LIN {X 0,Y 255.719,Z 484.142,A -85,B 0,C 180,E1 -18832.417,E2 -18832.417} C_VEL
LIN {X 0,Y 257.097,Z 472.751,A -85,B 0,C 180,E1 -18833.566,E2 -18833.566} C_VEL
LIN {X 0,Y 258.388,Z 459.153,A -85,B 0,C 180,E1 -18834.561,E2 -18834.561} C_VEL
LIN {X 0,Y 259.209,Z 446.518,A -85,B 0,C 180,E1 -18835.173,E2 -18835.173} C_VEL
LIN {X 0,Y 260.998,Z 385.807,A -85,B 0,C 180,E1 -18836.837,E2 -18836.837} C_VEL
LIN {X 0,Y 256.391,Z 351.056,A -85,B 0,C 180,E1 -18838.294,E2 -18838.294} C_VEL
LIN {X 0,Y 251.982,Z 338.318,A -85,B 0,C 180,E1 -18839.157,E2 -18839.157} C_VEL
LIN {X 0,Y 250.109,Z 329.208,A -85,B 0,C 180,E1 -18842.542,E2 -18842.542} C_VEL
LIN {X 0,Y 249.068,Z 324.462,A -85,B 0,C 180,E1 -18844.447,E2 -18844.447} C_VEL
LIN {X 0,Y 249.006,Z 324.47,A -85,B 0,C 180,E1 -18848.386,E2 -18848.386} C_VEL
LIN {X 0,Y 248.98,Z 324.473,A -85,B 0,C 180,E1 -18852.785,E2 -18852.785} C_VEL
LIN {X 0,Y 249.014,Z 324.467,A -85,B 0,C 180,E1 -18857.362,E2 -18857.362} C_VEL
LIN {X 0,Y 249.031,Z 324.461,A -85,B 0,C 180,E1 -18861.62,E2 -18861.62} C_VEL
LIN {X 0,Y 249.048,Z 324.46,A -85,B 0,C 180,E1 -18865.64,E2 -18865.64} C_VEL
LIN {X 0,Y 249.008,Z 324.466,A -85,B 0,C 180,E1 -18869.467,E2 -18869.467} C_VEL
LIN {X 0,Y 249.046,Z 324.462,A -85,B 0,C 180,E1 -18873.159,E2 -18873.159} C_VEL
LIN {X 0,Y 249.061,Z 324.459,A -85,B 0,C 180,E1 -18876.73,E2 -18876.73} C_VEL
LIN {X 0,Y 249.083,Z 324.443,A -85,B 0,C 180,E1 -18880.209,E2 -18880.209} C_VEL
LIN {X 0,Y 249.182,Z 324.446,A -85,B 0,C 180,E1 -18883.617,E2 -18883.617} C_VEL
LIN {X 0,Y 249.218,Z 324.438,A -85,B 0,C 180,E1 -18886.961,E2 -18886.961} C_VEL
LIN {X 0,Y 249.446,Z 324.399,A -85,B 0,C 180,E1 -18891.901,E2 -18891.901} C_VEL
LIN {X 0,Y 249.28,Z 324.429,A -85,B 0,C 180,E1 -18895.148,E2 -18895.148} C_VEL
LIN {X 0,Y 249.668,Z 324.38,A -85,B 0,C 180,E1 -18898.387,E2 -18898.387} C_VEL
LIN {X 0,Y 249.67,Z 324.37,A -85,B 0,C 180,E1 -18901.613,E2 -18901.613} C_VEL
LIN {X 0,Y 249.429,Z 324.411,A -85,B 0,C 180,E1 -18906.582,E2 -18906.582} C_VEL
LIN {X 0,Y 249.348,Z 324.422,A -85,B 0,C 180,E1 -18909.736,E2 -18909.736} C_VEL
LIN {X 0,Y 249.176,Z 324.427,A -85,B 0,C 180,E1 -18914.705,E2 -18914.705} C_VEL
LIN {X 0,Y 249.107,Z 324.445,A -85,B 0,C 180,E1 -18918.079,E2 -18918.079} C_VEL
LIN {X 0,Y 249.084,Z 324.456,A -85,B 0,C 180,E1 -18921.518,E2 -18921.518} C_VEL
LIN {X 0,Y 249.09,Z 324.445,A -85,B 0,C 180,E1 -18925.46,E2 -18925.46} C_VEL
LIN {X 0,Y 249.04,Z 324.447,A -85,B 0,C 180,E1 -18928.973,E2 -18928.973} C_VEL
LIN {X 0,Y 249.031,Z 324.459,A -85,B 0,C 180,E1 -18932.425,E2 -18932.425} C_VEL
LIN {X 0,Y 249.033,Z 324.454,A -85,B 0,C 180,E1 -18936.344,E2 -18936.344} C_VEL
LIN {X 0,Y 249.009,Z 324.459,A -85,B 0,C 180,E1 -18940.477,E2 -18940.477} C_VEL
LIN {X 0,Y 248.998,Z 324.464,A -85,B 0,C 180,E1 -18944.88,E2 -18944.88} C_VEL
LIN {X 0,Y 249.012,Z 324.455,A -85,B 0,C 180,E1 -18947.36,E2 -18947.36} C_VEL
LIN {X 0,Y 249.026,Z 324.464,A -85,B 0,C 180,E1 -18951.618,E2 -18951.618} C_VEL
LIN {X 0,Y 249.045,Z 324.453,A -85,B 0,C 180,E1 -18955.638,E2 -18955.638} C_VEL
LIN {X 0,Y 249.005,Z 324.465,A -85,B 0,C 180,E1 -18959.465,E2 -18959.465} C_VEL
LIN {X 0,Y 249.045,Z 324.462,A -85,B 0,C 180,E1 -18963.158,E2 -18963.158} C_VEL
LIN {X 0,Y 249.061,Z 324.463,A -85,B 0,C 180,E1 -18966.729,E2 -18966.729} C_VEL
LIN {X 0,Y 249.105,Z 324.457,A -85,B 0,C 180,E1 -18970.21,E2 -18970.21} C_VEL
LIN {X 0,Y 249.258,Z 324.58,A -85,B 0,C 180,E1 -18974.147,E2 -18974.147} C_VEL
LIN {X 0,Y 249.54,Z 325.958,A -85,B 0,C 180,E1 -18974.698,E2 -18974.698} C_VEL
LIN {X 0,Y 257.53,Z 346.854,A -85,B 0,C 180,E1 -18976.149,E2 -18976.149} C_VEL
LIN {X 0,Y 260.689,Z 356.803,A -85,B 0,C 180,E1 -18976.741,E2 -18976.741} C_VEL
LIN {X 0,Y 261.615,Z 362.917,A -85,B 0,C 180,E1 -18977.005,E2 -18977.005} C_VEL
LIN {X 0,Y 259.361,Z 433.833,A -85,B 0,C 180,E1 -18978.943,E2 -18978.943} C_VEL
LIN {X 0,Y 258.474,Z 447.221,A -85,B 0,C 180,E1 -18979.621,E2 -18979.621} C_VEL
LIN {X 0,Y 257.42,Z 459.695,A -85,B 0,C 180,E1 -18980.571,E2 -18980.571} C_VEL
LIN {X 0,Y 256.267,Z 470.812,A -85,B 0,C 180,E1 -18981.72,E2 -18981.72} C_VEL
LIN {X 0,Y 254.576,Z 482.837,A -85,B 0,C 180,E1 -18983.324,E2 -18983.324} C_VEL
LIN {X 0,Y 252.924,Z 493.895,A -85,B 0,C 180,E1 -18985.217,E2 -18985.217} C_VEL
LIN {X 0,Y 251.319,Z 503.079,A -85,B 0,C 180,E1 -18987.194,E2 -18987.194} C_VEL
LIN {X 0,Y 249.795,Z 512.013,A -85,B 0,C 180,E1 -18989.596,E2 -18989.596} C_VEL
LIN {X 0,Y 248.687,Z 519.181,A -85,B 0,C 180,E1 -18992.023,E2 -18992.023} C_VEL
LIN {X 0,Y 247.943,Z 524.03,A -85,B 0,C 180,E1 -18994.062,E2 -18994.062} C_VEL
LIN {X 0,Y 247.436,Z 528.724,A -85,B 0,C 180,E1 -18996.522,E2 -18996.522} C_VEL
LIN {X 0,Y 247.001,Z 532.318,A -85,B 0,C 180,E1 -18999.002,E2 -18999.002} C_VEL
LIN {X 0,Y 246.706,Z 534.889,A -85,B 0,C 180,E1 -19001.501,E2 -19001.501} C_VEL
LIN {X 0,Y 246.684,Z 536.663,A -85,B 0,C 180,E1 -19004.385,E2 -19004.385} C_VEL
LIN {X 0,Y 246.768,Z 537.151,A -85,B 0,C 180,E1 -19006.545,E2 -19006.545} C_VEL
LIN {X 0,Y 246.969,Z 537.091,A -85,B 0,C 180,E1 -19008.24,E2 -19008.24} C_VEL
LIN {X 0,Y 247.414,Z 536.36,A -85,B 0,C 180,E1 -19010.383,E2 -19010.383} C_VEL
LIN {X 0,Y 248.3,Z 534.267,A -85,B 0,C 180,E1 -19013.343,E2 -19013.343} C_VEL
LIN {X 0,Y 249.262,Z 531.781,A -85,B 0,C 180,E1 -19015.546,E2 -19015.546} C_VEL
LIN {X 0,Y 251.01,Z 527.278,A -85,B 0,C 180,E1 -19018.421,E2 -19018.421} C_VEL
LIN {X 0,Y 253.289,Z 520.981,A -85,B 0,C 180,E1 -19021.316,E2 -19021.316} C_VEL
LIN {X 0,Y 255.771,Z 513.958,A -85,B 0,C 180,E1 -19023.778,E2 -19023.778} C_VEL
LIN {X 0,Y 258.049,Z 506.62,A -85,B 0,C 180,E1 -19025.84,E2 -19025.84} C_VEL
LIN {X 0,Y 260.777,Z 497.786,A -85,B 0,C 180,E1 -19027.813,E2 -19027.813} C_VEL
LIN {X 0,Y 263.289,Z 488.607,A -85,B 0,C 180,E1 -19029.459,E2 -19029.459} C_VEL
LIN {X 0,Y 265.977,Z 477.163,A -85,B 0,C 180,E1 -19031.091,E2 -19031.091} C_VEL
LIN {X 0,Y 268.366,Z 465.176,A -85,B 0,C 180,E1 -19032.401,E2 -19032.401} C_VEL
LIN {X 0,Y 270.302,Z 452.398,A -85,B 0,C 180,E1 -19033.432,E2 -19033.432} C_VEL
LIN {X 0,Y 271.66,Z 439.162,A -85,B 0,C 180,E1 -19034.19,E2 -19034.19} C_VEL
LIN {X 0,Y 272.593,Z 424.235,A -85,B 0,C 180,E1 -19034.673,E2 -19034.673} C_VEL
LIN {X 0,Y 274.789,Z 373.279,A -85,B 0,C 180,E1 -19035.986,E2 -19035.986} C_VEL
LIN {X 0,Y 268.616,Z 359.848,A -85,B 0,C 180,E1 -19037.452,E2 -19037.452} C_VEL
LIN {X 0,Y 261.644,Z 346.658,A -85,B 0,C 180,E1 -19039.165,E2 -19039.165} C_VEL
LIN {X 0,Y 254.22,Z 334.263,A -85,B 0,C 180,E1 -19041.093,E2 -19041.093} C_VEL
LIN {X 0,Y 251.4,Z 329.949,A -85,B 0,C 180,E1 -19041.857,E2 -19041.857} C_VEL
LIN {X 0,Y 249.757,Z 326.866,A -85,B 0,C 180,E1 -19042.358,E2 -19042.358} C_VEL
LIN {X 0,Y 249.039,Z 324.465,A -85,B 0,C 180,E1 -19043.745,E2 -19043.745} C_VEL
LIN {X 0,Y 249.025,Z 324.45,A -85,B 0,C 180,E1 -19047.847,E2 -19047.847} C_VEL
LIN {X 0,Y 249.04,Z 324.458,A -85,B 0,C 180,E1 -19051.332,E2 -19051.332} C_VEL
LIN {X 0,Y 249.091,Z 324.451,A -85,B 0,C 180,E1 -19054.962,E2 -19054.962} C_VEL
LIN {X 0,Y 249.044,Z 324.455,A -85,B 0,C 180,E1 -19058.626,E2 -19058.626} C_VEL
LIN {X 0,Y 249.15,Z 324.446,A -85,B 0,C 180,E1 -19063.616,E2 -19063.616} C_VEL
LIN {X 0,Y 249.209,Z 324.441,A -85,B 0,C 180,E1 -19068.615,E2 -19068.615} C_VEL
LIN {X 0,Y 249.405,Z 324.401,A -85,B 0,C 180,E1 -19071.901,E2 -19071.901} C_VEL
LIN {X 0,Y 249.243,Z 324.433,A -85,B 0,C 180,E1 -19075.148,E2 -19075.148} C_VEL
LIN {X 0,Y 249.621,Z 324.384,A -85,B 0,C 180,E1 -19078.973,E2 -19078.973} C_VEL
LIN {X 0,Y 249.649,Z 324.372,A -85,B 0,C 180,E1 -19081.614,E2 -19081.614} C_VEL
LIN {X 0,Y 249.343,Z 324.416,A -85,B 0,C 180,E1 -19085.947,E2 -19085.947} C_VEL
LIN {X 0,Y 248.769,Z 324.485,A -85,B 0,C 180,E1 -19087.294,E2 -19087.294} C_VEL
LIN {X 0,Y 247.167,Z 324.688,A -85,B 0,C 180,E1 -19088.616,E2 -19088.616} C_VEL
LIN {X 0,Y 243.282,Z 325.174,A -85,B 0,C 180,E1 -19091.274,E2 -19091.274} C_VEL
LIN {X 0,Y 242.198,Z 325.297,A -85,B 0,C 180,E1 -19092.665,E2 -19092.665} C_VEL
LIN {X 0,Y 242.121,Z 325.305,A -85,B 0,C 180,E1 -19093.137,E2 -19093.137} C_VEL
LIN {X 0,Y 242.106,Z 325.316,A -85,B 0,C 180,E1 -19096.876,E2 -19096.876} C_VEL
LIN {X 0,Y 242.012,Z 325.332,A -85,B 0,C 180,E1 -19101.683,E2 -19101.683} C_VEL
LIN {X 0,Y 241.987,Z 325.34,A -85,B 0,C 180,E1 -19105.827,E2 -19105.827} C_VEL
LIN {X 0,Y 241.963,Z 325.347,A -85,B 0,C 180,E1 -19109.59,E2 -19109.59} C_VEL
LIN {X 0,Y 241.973,Z 325.345,A -85,B 0,C 180,E1 -19113.494,E2 -19113.494} C_VEL
LIN {X 0,Y 241.959,Z 325.345,A -85,B 0,C 180,E1 -19117.588,E2 -19117.588} C_VEL
LIN {X 0,Y 241.901,Z 325.336,A -85,B 0,C 180,E1 -19121.931,E2 -19121.931} C_VEL
LIN {X 0,Y 241.928,Z 325.445,A -85,B 0,C 180,E1 -19124.566,E2 -19124.566} C_VEL
LIN {X 0,Y 244.093,Z 332.594,A -85,B 0,C 180,E1 -19128.533,E2 -19128.533} C_VEL
LIN {X 0,Y 245.363,Z 336.886,A -85,B 0,C 180,E1 -19130.739,E2 -19130.739} C_VEL
LIN {X 0,Y 247.923,Z 341.395,A -85,B 0,C 180,E1 -19131.498,E2 -19131.498} C_VEL
LIN {X 0,Y 252.243,Z 349.01,A -85,B 0,C 180,E1 -19132.724,E2 -19132.724} C_VEL
LIN {X 0,Y 258.272,Z 360.24,A -85,B 0,C 180,E1 -19134.35,E2 -19134.35} C_VEL
LIN {X 0,Y 265.204,Z 375.094,A -85,B 0,C 180,E1 -19136.145,E2 -19136.145} C_VEL
LIN {X 0,Y 266.211,Z 378.364,A -85,B 0,C 180,E1 -19136.431,E2 -19136.431} C_VEL
LIN {X 0,Y 268.448,Z 392.441,A -85,B 0,C 180,E1 -19137.285,E2 -19137.285} C_VEL
LIN {X 0,Y 265.992,Z 446.475,A -85,B 0,C 180,E1 -19138.744,E2 -19138.744} C_VEL
LIN {X 0,Y 264.593,Z 460.076,A -85,B 0,C 180,E1 -19139.385,E2 -19139.385} C_VEL
LIN {X 0,Y 262.629,Z 472.258,A -85,B 0,C 180,E1 -19140.218,E2 -19140.218} C_VEL
LIN {X 0,Y 260.301,Z 484.181,A -85,B 0,C 180,E1 -19141.366,E2 -19141.366} C_VEL
LIN {X 0,Y 257.528,Z 495.6,A -85,B 0,C 180,E1 -19142.801,E2 -19142.801} C_VEL
LIN {X 0,Y 254.771,Z 505.898,A -85,B 0,C 180,E1 -19144.469,E2 -19144.469} C_VEL
LIN {X 0,Y 252.107,Z 514.351,A -85,B 0,C 180,E1 -19146.16,E2 -19146.16} C_VEL
LIN {X 0,Y 249.473,Z 522.167,A -85,B 0,C 180,E1 -19148.084,E2 -19148.084} C_VEL
LIN {X 0,Y 246.92,Z 529.825,A -85,B 0,C 180,E1 -19150.463,E2 -19150.463} C_VEL
LIN {X 0,Y 244.37,Z 536.91,A -85,B 0,C 180,E1 -19153.288,E2 -19153.288} C_VEL
LIN {X 0,Y 242.596,Z 541.655,A -85,B 0,C 180,E1 -19155.746,E2 -19155.746} C_VEL
LIN {X 0,Y 241.34,Z 545.309,A -85,B 0,C 180,E1 -19158.24,E2 -19158.24} C_VEL
LIN {X 0,Y 240.725,Z 547.212,A -85,B 0,C 180,E1 -19159.913,E2 -19159.913} C_VEL
LIN {X 0,Y 240.275,Z 548.673,A -85,B 0,C 180,E1 -19161.592,E2 -19161.592} C_VEL
LIN {X 0,Y 239.802,Z 550.385,A -85,B 0,C 180,E1 -19164.957,E2 -19164.957} C_VEL
LIN {X 0,Y 239.763,Z 550.671,A -85,B 0,C 180,E1 -19166.641,E2 -19166.641} C_VEL
LIN {X 0,Y 239.832,Z 550.555,A -85,B 0,C 180,E1 -19168.322,E2 -19168.322} C_VEL
LIN {X 0,Y 239.915,Z 550.015,A -85,B 0,C 180,E1 -19170.002,E2 -19170.002} C_VEL
LIN {X 0,Y 239.868,Z 549.078,A -85,B 0,C 180,E1 -19171.68,E2 -19171.68} C_VEL
LIN {X 0,Y 239.807,Z 547.737,A -85,B 0,C 180,E1 -19173.362,E2 -19173.362} C_VEL
LIN {X 0,Y 239.907,Z 544.883,A -85,B 0,C 180,E1 -19175.886,E2 -19175.886} C_VEL
LIN {X 0,Y 240.201,Z 540.977,A -85,B 0,C 180,E1 -19178.414,E2 -19178.414} C_VEL
LIN {X 0,Y 240.76,Z 535.915,A -85,B 0,C 180,E1 -19180.939,E2 -19180.939} C_VEL
LIN {X 0,Y 241.624,Z 529.527,A -85,B 0,C 180,E1 -19183.457,E2 -19183.457} C_VEL
LIN {X 0,Y 242.956,Z 521.508,A -85,B 0,C 180,E1 -19185.952,E2 -19185.952} C_VEL
LIN {X 0,Y 244.419,Z 513.328,A -85,B 0,C 180,E1 -19188.007,E2 -19188.007} C_VEL
LIN {X 0,Y 245.93,Z 503.3,A -85,B 0,C 180,E1 -19190.057,E2 -19190.057} C_VEL
LIN {X 0,Y 247.736,Z 492.021,A -85,B 0,C 180,E1 -19191.862,E2 -19191.862} C_VEL
LIN {X 0,Y 249.346,Z 480.953,A -85,B 0,C 180,E1 -19193.242,E2 -19193.242} C_VEL
LIN {X 0,Y 250.815,Z 468.678,A -85,B 0,C 180,E1 -19194.414,E2 -19194.414} C_VEL
LIN {X 0,Y 251.969,Z 455.818,A -85,B 0,C 180,E1 -19195.285,E2 -19195.285} C_VEL
LIN {X 0,Y 252.75,Z 442.198,A -85,B 0,C 180,E1 -19195.864,E2 -19195.864} C_VEL
LIN {X 0,Y 254.347,Z 386.316,A -85,B 0,C 180,E1 -19197.418,E2 -19197.418} C_VEL
LIN {X 0,Y 250.029,Z 353.01,A -85,B 0,C 180,E1 -19198.857,E2 -19198.857} C_VEL
LIN {X 0,Y 244.73,Z 338.103,A -85,B 0,C 180,E1 -19199.918,E2 -19199.918} C_VEL
LIN {X 0,Y 242.559,Z 327.821,A -85,B 0,C 180,E1 -19203.902,E2 -19203.902} C_VEL
LIN {X 0,Y 242.024,Z 325.336,A -85,B 0,C 180,E1 -19204.997,E2 -19204.997} C_VEL
LIN {X 0,Y 241.934,Z 325.35,A -85,B 0,C 180,E1 -19209.725,E2 -19209.725} C_VEL
LIN {X 0,Y 241.915,Z 325.355,A -85,B 0,C 180,E1 -19214.207,E2 -19214.207} C_VEL
LIN {X 0,Y 241.939,Z 325.351,A -85,B 0,C 180,E1 -19218.077,E2 -19218.077} C_VEL
LIN {X 0,Y 241.992,Z 325.341,A -85,B 0,C 180,E1 -19222.418,E2 -19222.418} C_VEL
LIN {X 0,Y 241.985,Z 325.342,A -85,B 0,C 180,E1 -19226.508,E2 -19226.508} C_VEL
LIN {X 0,Y 241.984,Z 325.342,A -85,B 0,C 180,E1 -19230.612,E2 -19230.612} C_VEL
LIN {X 0,Y 242.038,Z 325.333,A -85,B 0,C 180,E1 -19234.179,E2 -19234.179} C_VEL
LIN {X 0,Y 242.028,Z 325.329,A -85,B 0,C 180,E1 -19238.316,E2 -19238.316} C_VEL
LIN {X 0,Y 242.121,Z 325.322,A -85,B 0,C 180,E1 -19243.316,E2 -19243.316} C_VEL
LIN {X 0,Y 242.183,Z 325.308,A -85,B 0,C 180,E1 -19248.279,E2 -19248.279} C_VEL
LIN {X 0,Y 242.395,Z 325.274,A -85,B 0,C 180,E1 -19251.664,E2 -19251.664} C_VEL
LIN {X 0,Y 242.241,Z 325.306,A -85,B 0,C 180,E1 -19255.006,E2 -19255.006} C_VEL
LIN {X 0,Y 242.628,Z 325.257,A -85,B 0,C 180,E1 -19258.34,E2 -19258.34} C_VEL
LIN {X 0,Y 242.63,Z 325.245,A -85,B 0,C 180,E1 -19261.659,E2 -19261.659} C_VEL
LIN {X 0,Y 242.407,Z 325.288,A -85,B 0,C 180,E1 -19266.659,E2 -19266.659} C_VEL
LIN {X 0,Y 242.272,Z 325.305,A -85,B 0,C 180,E1 -19270.023,E2 -19270.023} C_VEL
LIN {X 0,Y 242.131,Z 325.302,A -85,B 0,C 180,E1 -19275.143,E2 -19275.143} C_VEL
LIN {X 0,Y 242.046,Z 325.327,A -85,B 0,C 180,E1 -19278.626,E2 -19278.626} C_VEL
LIN {X 0,Y 242.007,Z 325.337,A -85,B 0,C 180,E1 -19282.18,E2 -19282.18} C_VEL
LIN {X 0,Y 242.036,Z 325.321,A -85,B 0,C 180,E1 -19285.82,E2 -19285.82} C_VEL
LIN {X 0,Y 241.972,Z 325.332,A -85,B 0,C 180,E1 -19289.588,E2 -19289.588} C_VEL
LIN {X 0,Y 241.983,Z 325.341,A -85,B 0,C 180,E1 -19293.492,E2 -19293.492} C_VEL
LIN {X 0,Y 241.989,Z 325.325,A -85,B 0,C 180,E1 -19297.581,E2 -19297.581} C_VEL
LIN {X 0,Y 241.94,Z 325.346,A -85,B 0,C 180,E1 -19301.921,E2 -19301.921} C_VEL
LIN {X 0,Y 241.93,Z 325.337,A -85,B 0,C 180,E1 -19306.572,E2 -19306.572} C_VEL
LIN {X 0,Y 241.958,Z 325.346,A -85,B 0,C 180,E1 -19310.28,E2 -19310.28} C_VEL
LIN {X 0,Y 241.987,Z 325.333,A -85,B 0,C 180,E1 -19314.488,E2 -19314.488} C_VEL
LIN {X 0,Y 241.956,Z 325.347,A -85,B 0,C 180,E1 -19318.476,E2 -19318.476} C_VEL
LIN {X 0,Y 241.976,Z 325.344,A -85,B 0,C 180,E1 -19322.307,E2 -19322.307} C_VEL
LIN {X 0,Y 242.039,Z 325.335,A -85,B 0,C 180,E1 -19326.013,E2 -19326.013} C_VEL
LIN {X 0,Y 242.034,Z 325.337,A -85,B 0,C 180,E1 -19329.606,E2 -19329.606} C_VEL
LIN {X 0,Y 242.174,Z 325.41,A -85,B 0,C 180,E1 -19333.616,E2 -19333.616} C_VEL
LIN {X 0,Y 242.324,Z 326.153,A -85,B 0,C 180,E1 -19333.924,E2 -19333.924} C_VEL
LIN {X 0,Y 250.238,Z 346.246,A -85,B 0,C 180,E1 -19335.415,E2 -19335.415} C_VEL
LIN {X 0,Y 254.218,Z 358.37,A -85,B 0,C 180,E1 -19336.181,E2 -19336.181} C_VEL
LIN {X 0,Y 255.039,Z 363.888,A -85,B 0,C 180,E1 -19336.428,E2 -19336.428} C_VEL
LIN {X 0,Y 252.719,Z 434.063,A -85,B 0,C 180,E1 -19338.391,E2 -19338.391} C_VEL
LIN {X 0,Y 251.799,Z 447.489,A -85,B 0,C 180,E1 -19339.088,E2 -19339.088} C_VEL
LIN {X 0,Y 250.757,Z 459.388,A -85,B 0,C 180,E1 -19340.012,E2 -19340.012} C_VEL
LIN {X 0,Y 249.462,Z 471.44,A -85,B 0,C 180,E1 -19341.289,E2 -19341.289} C_VEL
LIN {X 0,Y 247.78,Z 482.955,A -85,B 0,C 180,E1 -19342.867,E2 -19342.867} C_VEL
LIN {X 0,Y 246.116,Z 493.358,A -85,B 0,C 180,E1 -19344.674,E2 -19344.674} C_VEL
LIN {X 0,Y 244.491,Z 502.683,A -85,B 0,C 180,E1 -19346.703,E2 -19346.703} C_VEL
LIN {X 0,Y 242.914,Z 511.712,A -85,B 0,C 180,E1 -19349.17,E2 -19349.17} C_VEL
LIN {X 0,Y 241.731,Z 518.983,A -85,B 0,C 180,E1 -19351.665,E2 -19351.665} C_VEL
LIN {X 0,Y 240.831,Z 524.793,A -85,B 0,C 180,E1 -19354.182,E2 -19354.182} C_VEL
LIN {X 0,Y 240.291,Z 529.359,A -85,B 0,C 180,E1 -19356.717,E2 -19356.717} C_VEL
LIN {X 0,Y 240.001,Z 531.774,A -85,B 0,C 180,E1 -19358.418,E2 -19358.418} C_VEL
LIN {X 0,Y 239.739,Z 533.761,A -85,B 0,C 180,E1 -19360.129,E2 -19360.129} C_VEL
LIN {X 0,Y 239.582,Z 535.318,A -85,B 0,C 180,E1 -19361.848,E2 -19361.848} C_VEL
LIN {X 0,Y 239.605,Z 536.865,A -85,B 0,C 180,E1 -19364.548,E2 -19364.548} C_VEL
LIN {X 0,Y 239.712,Z 537.382,A -85,B 0,C 180,E1 -19367.047,E2 -19367.047} C_VEL
LIN {X 0,Y 239.962,Z 537.232,A -85,B 0,C 180,E1 -19368.792,E2 -19368.792} C_VEL
LIN {X 0,Y 240.379,Z 536.58,A -85,B 0,C 180,E1 -19370.678,E2 -19370.678} C_VEL
LIN {X 0,Y 241.46,Z 534.213,A -85,B 0,C 180,E1 -19374.045,E2 -19374.045} C_VEL
LIN {X 0,Y 242.702,Z 531.284,A -85,B 0,C 180,E1 -19376.574,E2 -19376.574} C_VEL
LIN {X 0,Y 244.455,Z 526.964,A -85,B 0,C 180,E1 -19379.256,E2 -19379.256} C_VEL
LIN {X 0,Y 246.563,Z 521.484,A -85,B 0,C 180,E1 -19381.823,E2 -19381.823} C_VEL
LIN {X 0,Y 249.129,Z 514.543,A -85,B 0,C 180,E1 -19384.345,E2 -19384.345} C_VEL
LIN {X 0,Y 251.503,Z 507.387,A -85,B 0,C 180,E1 -19386.426,E2 -19386.426} C_VEL
LIN {X 0,Y 254.348,Z 498.71,A -85,B 0,C 180,E1 -19388.439,E2 -19388.439} C_VEL
LIN {X 0,Y 257.098,Z 489.107,A -85,B 0,C 180,E1 -19390.219,E2 -19390.219} C_VEL
LIN {X 0,Y 259.74,Z 478.482,A -85,B 0,C 180,E1 -19391.78,E2 -19391.78} C_VEL
LIN {X 0,Y 262.196,Z 466.802,A -85,B 0,C 180,E1 -19393.116,E2 -19393.116} C_VEL
LIN {X 0,Y 264.127,Z 455.272,A -85,B 0,C 180,E1 -19394.117,E2 -19394.117} C_VEL
LIN {X 0,Y 265.681,Z 441.84,A -85,B 0,C 180,E1 -19394.948,E2 -19394.948} C_VEL
LIN {X 0,Y 266.64,Z 428.837,A -85,B 0,C 180,E1 -19395.449,E2 -19395.449} C_VEL
LIN {X 0,Y 269.139,Z 376.062,A -85,B 0,C 180,E1 -19396.815,E2 -19396.815} C_VEL
LIN {X 0,Y 267.651,Z 372.135,A -85,B 0,C 180,E1 -19397.199,E2 -19397.199} C_VEL
LIN {X 0,Y 260.471,Z 357.236,A -85,B 0,C 180,E1 -19399.005,E2 -19399.005} C_VEL
LIN {X 0,Y 253.369,Z 344.62,A -85,B 0,C 180,E1 -19400.873,E2 -19400.873} C_VEL
LIN {X 0,Y 247.499,Z 335.143,A -85,B 0,C 180,E1 -19402.509,E2 -19402.509} C_VEL
LIN {X 0,Y 245.051,Z 331.288,A -85,B 0,C 180,E1 -19403.225,E2 -19403.225} C_VEL
LIN {X 0,Y 242.452,Z 327.124,A -85,B 0,C 180,E1 -19404.058,E2 -19404.058} C_VEL
LIN {X 0,Y 241.996,Z 325.318,A -85,B 0,C 180,E1 -19405.127,E2 -19405.127} C_VEL
LIN {X 0,Y 241.946,Z 325.342,A -85,B 0,C 180,E1 -19408.476,E2 -19408.476} C_VEL
LIN {X 0,Y 241.959,Z 325.347,A -85,B 0,C 180,E1 -19412.307,E2 -19412.307} C_VEL
LIN {X 0,Y 242.013,Z 325.34,A -85,B 0,C 180,E1 -19416.012,E2 -19416.012} C_VEL
LIN {X 0,Y 241.976,Z 325.343,A -85,B 0,C 180,E1 -19419.603,E2 -19419.603} C_VEL
LIN {X 0,Y 242.097,Z 325.322,A -85,B 0,C 180,E1 -19423.324,E2 -19423.324} C_VEL
LIN {X 0,Y 242.143,Z 325.317,A -85,B 0,C 180,E1 -19428.278,E2 -19428.278} C_VEL
LIN {X 0,Y 242.359,Z 325.278,A -85,B 0,C 180,E1 -19431.664,E2 -19431.664} C_VEL
LIN {X 0,Y 242.386,Z 325.289,A -85,B 0,C 180,E1 -19433.34,E2 -19433.34} C_VEL
LIN {X 0,Y 242.597,Z 325.258,A -85,B 0,C 180,E1 -19438.34,E2 -19438.34} C_VEL
LIN {X 0,Y 242.609,Z 325.248,A -85,B 0,C 180,E1 -19441.66,E2 -19441.66} C_VEL
LIN {X 0,Y 242.39,Z 325.278,A -85,B 0,C 180,E1 -19446.66,E2 -19446.66} C_VEL
LIN {X 0,Y 242.259,Z 325.304,A -85,B 0,C 180,E1 -19450.024,E2 -19450.024} C_VEL
LIN {X 0,Y 242.121,Z 325.305,A -85,B 0,C 180,E1 -19453.137,E2 -19453.137} C_VEL
LIN {X 0,Y 241.464,Z 325.396,A -85,B 0,C 180,E1 -19454.525,E2 -19454.525} C_VEL
LIN {X 0,Y 238.549,Z 325.76,A -85,B 0,C 180,E1 -19456.786,E2 -19456.786} C_VEL
LIN {X 0,Y 236.071,Z 326.063,A -85,B 0,C 180,E1 -19458.629,E2 -19458.629} C_VEL
LIN {X 0,Y 235.031,Z 326.203,A -85,B 0,C 180,E1 -19460.061,E2 -19460.061} C_VEL
LIN {X 0,Y 234.96,Z 326.208,A -85,B 0,C 180,E1 -19460.547,E2 -19460.547} C_VEL
LIN {X 0,Y 234.918,Z 326.218,A -85,B 0,C 180,E1 -19464.762,E2 -19464.762} C_VEL
LIN {X 0,Y 234.894,Z 326.217,A -85,B 0,C 180,E1 -19468.602,E2 -19468.602} C_VEL
LIN {X 0,Y 234.935,Z 326.218,A -85,B 0,C 180,E1 -19473.115,E2 -19473.115} C_VEL
LIN {X 0,Y 234.901,Z 326.223,A -85,B 0,C 180,E1 -19476.755,E2 -19476.755} C_VEL
LIN {X 0,Y 234.907,Z 326.217,A -85,B 0,C 180,E1 -19478.937,E2 -19478.937} C_VEL
LIN {X 0,Y 234.846,Z 326.254,A -85,B 0,C 180,E1 -19482.973,E2 -19482.973} C_VEL
LIN {X 0,Y 236.943,Z 333.006,A -85,B 0,C 180,E1 -19486.986,E2 -19486.986} C_VEL
LIN {X 0,Y 238.036,Z 336.737,A -85,B 0,C 180,E1 -19488.961,E2 -19488.961} C_VEL
LIN {X 0,Y 240.812,Z 341.34,A -85,B 0,C 180,E1 -19489.849,E2 -19489.849} C_VEL
LIN {X 0,Y 245.278,Z 348.905,A -85,B 0,C 180,E1 -19491.209,E2 -19491.209} C_VEL
LIN {X 0,Y 250.995,Z 359.266,A -85,B 0,C 180,E1 -19492.859,E2 -19492.859} C_VEL
LIN {X 0,Y 258.542,Z 374.896,A -85,B 0,C 180,E1 -19494.933,E2 -19494.933} C_VEL
LIN {X 0,Y 260.834,Z 380.697,A -85,B 0,C 180,E1 -19495.565,E2 -19495.565} C_VEL
LIN {X 0,Y 262.83,Z 393.388,A -85,B 0,C 180,E1 -19496.365,E2 -19496.365} C_VEL
LIN {X 0,Y 260.35,Z 445.928,A -85,B 0,C 180,E1 -19497.804,E2 -19497.804} C_VEL
LIN {X 0,Y 258.909,Z 459.585,A -85,B 0,C 180,E1 -19498.45,E2 -19498.45} C_VEL
LIN {X 0,Y 256.941,Z 471.451,A -85,B 0,C 180,E1 -19499.261,E2 -19499.261} C_VEL
LIN {X 0,Y 254.514,Z 483.556,A -85,B 0,C 180,E1 -19500.425,E2 -19500.425} C_VEL
LIN {X 0,Y 251.651,Z 495.05,A -85,B 0,C 180,E1 -19501.885,E2 -19501.885} C_VEL
LIN {X 0,Y 248.708,Z 505.414,A -85,B 0,C 180,E1 -19503.574,E2 -19503.574} C_VEL
LIN {X 0,Y 245.652,Z 514.783,A -85,B 0,C 180,E1 -19505.493,E2 -19505.493} C_VEL
LIN {X 0,Y 242.414,Z 523.833,A -85,B 0,C 180,E1 -19507.86,E2 -19507.86} C_VEL
LIN {X 0,Y 239.85,Z 531.143,A -85,B 0,C 180,E1 -19510.309,E2 -19510.309} C_VEL
LIN {X 0,Y 237.582,Z 537.035,A -85,B 0,C 180,E1 -19512.795,E2 -19512.795} C_VEL
LIN {X 0,Y 235.711,Z 541.708,A -85,B 0,C 180,E1 -19515.321,E2 -19515.321} C_VEL
LIN {X 0,Y 234.375,Z 545.296,A -85,B 0,C 180,E1 -19517.885,E2 -19517.885} C_VEL
LIN {X 0,Y 233.724,Z 547.16,A -85,B 0,C 180,E1 -19519.608,E2 -19519.608} C_VEL
LIN {X 0,Y 232.905,Z 549.59,A -85,B 0,C 180,E1 -19523.069,E2 -19523.069} C_VEL
LIN {X 0,Y 232.672,Z 550.483,A -85,B 0,C 180,E1 -19526.538,E2 -19526.538} C_VEL
LIN {X 0,Y 232.743,Z 550.315,A -85,B 0,C 180,E1 -19528.271,E2 -19528.271} C_VEL
LIN {X 0,Y 232.846,Z 549.747,A -85,B 0,C 180,E1 -19530.002,E2 -19530.002} C_VEL
LIN {X 0,Y 232.778,Z 548.78,A -85,B 0,C 180,E1 -19531.732,E2 -19531.732} C_VEL
LIN {X 0,Y 232.759,Z 545.989,A -85,B 0,C 180,E1 -19534.85,E2 -19534.85} C_VEL
LIN {X 0,Y 233.004,Z 541.967,A -85,B 0,C 180,E1 -19537.802,E2 -19537.802} C_VEL
LIN {X 0,Y 233.496,Z 537.227,A -85,B 0,C 180,E1 -19540.406,E2 -19540.406} C_VEL
LIN {X 0,Y 234.502,Z 530.075,A -85,B 0,C 180,E1 -19543.432,E2 -19543.432} C_VEL
LIN {X 0,Y 235.853,Z 522.29,A -85,B 0,C 180,E1 -19546.001,E2 -19546.001} C_VEL
LIN {X 0,Y 237.49,Z 513.193,A -85,B 0,C 180,E1 -19548.378,E2 -19548.378} C_VEL
LIN {X 0,Y 239.01,Z 503.533,A -85,B 0,C 180,E1 -19550.416,E2 -19550.416} C_VEL
LIN {X 0,Y 240.616,Z 493.635,A -85,B 0,C 180,E1 -19552.091,E2 -19552.091} C_VEL
LIN {X 0,Y 242.351,Z 483.078,A -85,B 0,C 180,E1 -19553.501,E2 -19553.501} C_VEL
LIN {X 0,Y 243.946,Z 470.304,A -85,B 0,C 180,E1 -19554.807,E2 -19554.807} C_VEL
LIN {X 0,Y 245.149,Z 457.51,A -85,B 0,C 180,E1 -19555.755,E2 -19555.755} C_VEL
LIN {X 0,Y 246.021,Z 445.318,A -85,B 0,C 180,E1 -19556.34,E2 -19556.34} C_VEL
LIN {X 0,Y 247.789,Z 387.009,A -85,B 0,C 180,E1 -19558.018,E2 -19558.018} C_VEL
LIN {X 0,Y 243.752,Z 355.347,A -85,B 0,C 180,E1 -19559.425,E2 -19559.425} C_VEL
LIN {X 0,Y 238.106,Z 339.877,A -85,B 0,C 180,E1 -19560.541,E2 -19560.541} C_VEL
LIN {X 0,Y 237.468,Z 337.867,A -85,B 0,C 180,E1 -19560.734,E2 -19560.734} C_VEL
LIN {X 0,Y 235.437,Z 328.392,A -85,B 0,C 180,E1 -19564.554,E2 -19564.554} C_VEL
LIN {X 0,Y 234.955,Z 326.215,A -85,B 0,C 180,E1 -19565.521,E2 -19565.521} C_VEL
LIN {X 0,Y 234.916,Z 326.223,A -85,B 0,C 180,E1 -19568.936,E2 -19568.936} C_VEL
LIN {X 0,Y 234.879,Z 326.231,A -85,B 0,C 180,E1 -19574.1,E2 -19574.1} C_VEL
LIN {X 0,Y 234.887,Z 326.228,A -85,B 0,C 180,E1 -19578.832,E2 -19578.832} C_VEL
LIN {X 0,Y 234.923,Z 326.22,A -85,B 0,C 180,E1 -19581.079,E2 -19581.079} C_VEL
LIN {X 0,Y 234.932,Z 326.219,A -85,B 0,C 180,E1 -19585.362,E2 -19585.362} C_VEL
LIN {X 0,Y 234.905,Z 326.223,A -85,B 0,C 180,E1 -19589.428,E2 -19589.428} C_VEL
LIN {X 0,Y 234.975,Z 326.213,A -85,B 0,C 180,E1 -19593.807,E2 -19593.807} C_VEL
LIN {X 0,Y 234.993,Z 326.202,A -85,B 0,C 180,E1 -19598.968,E2 -19598.968} C_VEL
LIN {X 0,Y 235.061,Z 326.2,A -85,B 0,C 180,E1 -19603.092,E2 -19603.092} C_VEL
LIN {X 0,Y 235.115,Z 326.19,A -85,B 0,C 180,E1 -19607.922,E2 -19607.922} C_VEL
LIN {X 0,Y 235.328,Z 326.151,A -85,B 0,C 180,E1 -19611.412,E2 -19611.412} C_VEL
LIN {X 0,Y 235.366,Z 326.156,A -85,B 0,C 180,E1 -19613.14,E2 -19613.14} C_VEL
LIN {X 0,Y 235.587,Z 326.134,A -85,B 0,C 180,E1 -19618.29,E2 -19618.29} C_VEL
LIN {X 0,Y 235.588,Z 326.12,A -85,B 0,C 180,E1 -19621.709,E2 -19621.709} C_VEL
LIN {X 0,Y 235.359,Z 326.165,A -85,B 0,C 180,E1 -19626.86,E2 -19626.86} C_VEL
LIN {X 0,Y 235.219,Z 326.185,A -85,B 0,C 180,E1 -19630.327,E2 -19630.327} C_VEL
LIN {X 0,Y 235.078,Z 326.18,A -85,B 0,C 180,E1 -19635.608,E2 -19635.608} C_VEL
LIN {X 0,Y 234.988,Z 326.211,A -85,B 0,C 180,E1 -19639.207,E2 -19639.207} C_VEL
LIN {X 0,Y 234.95,Z 326.218,A -85,B 0,C 180,E1 -19642.884,E2 -19642.884} C_VEL
LIN {X 0,Y 234.949,Z 326.2,A -85,B 0,C 180,E1 -19646.659,E2 -19646.659} C_VEL
LIN {X 0,Y 234.903,Z 326.214,A -85,B 0,C 180,E1 -19650.571,E2 -19650.571} C_VEL
LIN {X 0,Y 234.93,Z 326.215,A -85,B 0,C 180,E1 -19654.638,E2 -19654.638} C_VEL
LIN {X 0,Y 234.945,Z 326.199,A -85,B 0,C 180,E1 -19658.943,E2 -19658.943} C_VEL
LIN {X 0,Y 234.888,Z 326.225,A -85,B 0,C 180,E1 -19663.485,E2 -19663.485} C_VEL
LIN {X 0,Y 234.883,Z 326.214,A -85,B 0,C 180,E1 -19666.511,E2 -19666.511} C_VEL
LIN {X 0,Y 234.92,Z 326.22,A -85,B 0,C 180,E1 -19671.077,E2 -19671.077} C_VEL
LIN {X 0,Y 234.931,Z 326.21,A -85,B 0,C 180,E1 -19675.36,E2 -19675.36} C_VEL
LIN {X 0,Y 234.902,Z 326.222,A -85,B 0,C 180,E1 -19679.426,E2 -19679.426} C_VEL
LIN {X 0,Y 234.971,Z 326.215,A -85,B 0,C 180,E1 -19683.805,E2 -19683.805} C_VEL
LIN {X 0,Y 234.998,Z 326.215,A -85,B 0,C 180,E1 -19688.967,E2 -19688.967} C_VEL
LIN {X 0,Y 235.121,Z 326.379,A -85,B 0,C 180,E1 -19693.107,E2 -19693.107} C_VEL
LIN {X 0,Y 236.293,Z 329.307,A -85,B 0,C 180,E1 -19693.36,E2 -19693.36} C_VEL
LIN {X 0,Y 242.991,Z 345.81,A -85,B 0,C 180,E1 -19694.65,E2 -19694.65} C_VEL
LIN {X 0,Y 247.745,Z 359.842,A -85,B 0,C 180,E1 -19695.589,E2 -19695.589} C_VEL
LIN {X 0,Y 248.492,Z 365.668,A -85,B 0,C 180,E1 -19695.846,E2 -19695.846} C_VEL
LIN {X 0,Y 246.093,Z 434.425,A -85,B 0,C 180,E1 -19697.815,E2 -19697.815} C_VEL
LIN {X 0,Y 245.133,Z 447.764,A -85,B 0,C 180,E1 -19698.526,E2 -19698.526} C_VEL
LIN {X 0,Y 244.003,Z 460.193,A -85,B 0,C 180,E1 -19699.523,E2 -19699.523} C_VEL
LIN {X 0,Y 242.668,Z 472.068,A -85,B 0,C 180,E1 -19700.833,E2 -19700.833} C_VEL
LIN {X 0,Y 240.977,Z 483.236,A -85,B 0,C 180,E1 -19702.41,E2 -19702.41} C_VEL
LIN {X 0,Y 239.202,Z 493.845,A -85,B 0,C 180,E1 -19704.308,E2 -19704.308} C_VEL
LIN {X 0,Y 237.7,Z 502.277,A -85,B 0,C 180,E1 -19706.184,E2 -19706.184} C_VEL
LIN {X 0,Y 236.028,Z 511.414,A -85,B 0,C 180,E1 -19708.719,E2 -19708.719} C_VEL
LIN {X 0,Y 234.756,Z 518.774,A -85,B 0,C 180,E1 -19711.285,E2 -19711.285} C_VEL
LIN {X 0,Y 233.906,Z 523.765,A -85,B 0,C 180,E1 -19713.444,E2 -19713.444} C_VEL
LIN {X 0,Y 233.315,Z 528.948,A -85,B 0,C 180,E1 -19716.263,E2 -19716.263} C_VEL
LIN {X 0,Y 232.856,Z 532.321,A -85,B 0,C 180,E1 -19718.678,E2 -19718.678} C_VEL
LIN {X 0,Y 232.593,Z 534.254,A -85,B 0,C 180,E1 -19720.444,E2 -19720.444} C_VEL
LIN {X 0,Y 232.479,Z 535.706,A -85,B 0,C 180,E1 -19722.215,E2 -19722.215} C_VEL
LIN {X 0,Y 232.502,Z 537.059,A -85,B 0,C 180,E1 -19724.697,E2 -19724.697} C_VEL
LIN {X 0,Y 232.676,Z 537.593,A -85,B 0,C 180,E1 -19727.579,E2 -19727.579} C_VEL
LIN {X 0,Y 233.348,Z 536.802,A -85,B 0,C 180,E1 -19730.988,E2 -19730.988} C_VEL
LIN {X 0,Y 233.955,Z 535.663,A -85,B 0,C 180,E1 -19732.985,E2 -19732.985} C_VEL
LIN {X 0,Y 234.677,Z 534.124,A -85,B 0,C 180,E1 -19734.786,E2 -19734.786} C_VEL
LIN {X 0,Y 236.112,Z 530.958,A -85,B 0,C 180,E1 -19737.473,E2 -19737.473} C_VEL
LIN {X 0,Y 237.956,Z 526.638,A -85,B 0,C 180,E1 -19740.137,E2 -19740.137} C_VEL
LIN {X 0,Y 240.254,Z 521.03,A -85,B 0,C 180,E1 -19742.761,E2 -19742.761} C_VEL
LIN {X 0,Y 242.974,Z 513.939,A -85,B 0,C 180,E1 -19745.343,E2 -19745.343} C_VEL
LIN {X 0,Y 245.562,Z 506.619,A -85,B 0,C 180,E1 -19747.456,E2 -19747.456} C_VEL
LIN {X 0,Y 248.838,Z 496.647,A -85,B 0,C 180,E1 -19749.715,E2 -19749.715} C_VEL
LIN {X 0,Y 251.884,Z 486.384,A -85,B 0,C 180,E1 -19751.534,E2 -19751.534} C_VEL
LIN {X 0,Y 254.592,Z 475.258,A -85,B 0,C 180,E1 -19753.094,E2 -19753.094} C_VEL
LIN {X 0,Y 257.135,Z 462.892,A -85,B 0,C 180,E1 -19754.4,E2 -19754.4} C_VEL
LIN {X 0,Y 259.086,Z 450.174,A -85,B 0,C 180,E1 -19755.4,E2 -19755.4} C_VEL
LIN {X 0,Y 260.397,Z 437.567,A -85,B 0,C 180,E1 -19756.075,E2 -19756.075} C_VEL
LIN {X 0,Y 261.475,Z 420.375,A -85,B 0,C 180,E1 -19756.596,E2 -19756.596} C_VEL
LIN {X 0,Y 263.49,Z 377.694,A -85,B 0,C 180,E1 -19757.728,E2 -19757.728} C_VEL
LIN {X 0,Y 256.428,Z 362.633,A -85,B 0,C 180,E1 -19759.583,E2 -19759.583} C_VEL
LIN {X 0,Y 249.291,Z 349.644,A -85,B 0,C 180,E1 -19761.539,E2 -19761.539} C_VEL
LIN {X 0,Y 243.526,Z 340.22,A -85,B 0,C 180,E1 -19763.214,E2 -19763.214} C_VEL
LIN {X 0,Y 240.934,Z 336.178,A -85,B 0,C 180,E1 -19764.004,E2 -19764.004} C_VEL
LIN {X 0,Y 238.176,Z 332.019,A -85,B 0,C 180,E1 -19764.873,E2 -19764.873} C_VEL
LIN {X 0,Y 235.444,Z 328.019,A -85,B 0,C 180,E1 -19765.765,E2 -19765.765} C_VEL
LIN {X 0,Y 235.195,Z 327.362,A -85,B 0,C 180,E1 -19765.934,E2 -19765.934} C_VEL
LIN {X 0,Y 234.945,Z 326.192,A -85,B 0,C 180,E1 -19766.757,E2 -19766.757} C_VEL
LIN {X 0,Y 234.893,Z 326.22,A -85,B 0,C 180,E1 -19771.399,E2 -19771.399} C_VEL
LIN {X 0,Y 234.943,Z 326.215,A -85,B 0,C 180,E1 -19775.242,E2 -19775.242} C_VEL
LIN {X 0,Y 234.931,Z 326.215,A -85,B 0,C 180,E1 -19778.963,E2 -19778.963} C_VEL
LIN {X 0,Y 235.041,Z 326.198,A -85,B 0,C 180,E1 -19783.098,E2 -19783.098} C_VEL
LIN {X 0,Y 235.075,Z 326.194,A -85,B 0,C 180,E1 -19787.92,E2 -19787.92} C_VEL
LIN {X 0,Y 235.295,Z 326.157,A -85,B 0,C 180,E1 -19791.411,E2 -19791.411} C_VEL
LIN {X 0,Y 235.337,Z 326.163,A -85,B 0,C 180,E1 -19793.14,E2 -19793.14} C_VEL
LIN {X 0,Y 235.556,Z 326.135,A -85,B 0,C 180,E1 -19798.291,E2 -19798.291} C_VEL
LIN {X 0,Y 235.567,Z 326.125,A -85,B 0,C 180,E1 -19801.71,E2 -19801.71} C_VEL
LIN {X 0,Y 235.342,Z 326.154,A -85,B 0,C 180,E1 -19806.861,E2 -19806.861} C_VEL
LIN {X 0,Y 235.205,Z 326.184,A -85,B 0,C 180,E1 -19810.328,E2 -19810.328} C_VEL
LIN {X 0,Y 235.079,Z 326.199,A -85,B 0,C 180,E1 -19815.609,E2 -19815.609} C_VEL
LIN {X 0,Y 234.986,Z 326.198,A -85,B 0,C 180,E1 -19819.208,E2 -19819.208} C_VEL
LIN {X 0,Y 234.96,Z 326.208,A -85,B 0,C 180,E1 -19820.547,E2 -19820.547} C_VEL
LIN {X 0,Y 234.318,Z 326.298,A -85,B 0,C 180,E1 -19821.978,E2 -19821.978} C_VEL
LIN {X 0,Y 231.442,Z 326.653,A -85,B 0,C 180,E1 -19824.311,E2 -19824.311} C_VEL
LIN {X 0,Y 228.973,Z 326.958,A -85,B 0,C 180,E1 -19826.213,E2 -19826.213} C_VEL
LIN {X 0,Y 227.908,Z 327.083,A -85,B 0,C 180,E1 -19827.692,E2 -19827.692} C_VEL
LIN {X 0,Y 227.82,Z 327.094,A -85,B 0,C 180,E1 -19828.193,E2 -19828.193} C_VEL
LIN {X 0,Y 227.85,Z 327.092,A -85,B 0,C 180,E1 -19831.626,E2 -19831.626} C_VEL
LIN {X 0,Y 227.856,Z 327.094,A -85,B 0,C 180,E1 -19835.877,E2 -19835.877} C_VEL
LIN {X 0,Y 227.793,Z 327.112,A -85,B 0,C 180,E1 -19840.384,E2 -19840.384} C_VEL
LIN {X 0,Y 227.822,Z 327.139,A -85,B 0,C 180,E1 -19841.279,E2 -19841.279} C_VEL
LIN {X 0,Y 230.074,Z 334.409,A -85,B 0,C 180,E1 -19845.877,E2 -19845.877} C_VEL
LIN {X 0,Y 230.695,Z 336.446,A -85,B 0,C 180,E1 -19846.983,E2 -19846.983} C_VEL
LIN {X 0,Y 233.297,Z 340.785,A -85,B 0,C 180,E1 -19847.9,E2 -19847.9} C_VEL
LIN {X 0,Y 234.864,Z 343.196,A -85,B 0,C 180,E1 -19848.426,E2 -19848.426} C_VEL
LIN {X 0,Y 238.736,Z 349.538,A -85,B 0,C 180,E1 -19849.69,E2 -19849.69} C_VEL
LIN {X 0,Y 243.68,Z 358.252,A -85,B 0,C 180,E1 -19851.226,E2 -19851.226} C_VEL
LIN {X 0,Y 250.347,Z 371.44,A -85,B 0,C 180,E1 -19853.193,E2 -19853.193} C_VEL
LIN {X 0,Y 255.49,Z 382.919,A -85,B 0,C 180,E1 -19854.646,E2 -19854.646} C_VEL
LIN {X 0,Y 257.278,Z 394.385,A -85,B 0,C 180,E1 -19855.401,E2 -19855.401} C_VEL
LIN {X 0,Y 254.693,Z 446.411,A -85,B 0,C 180,E1 -19856.861,E2 -19856.861} C_VEL
LIN {X 0,Y 253.169,Z 460,A -85,B 0,C 180,E1 -19857.523,E2 -19857.523} C_VEL
LIN {X 0,Y 251.127,Z 471.774,A -85,B 0,C 180,E1 -19858.352,E2 -19858.352} C_VEL
LIN {X 0,Y 248.765,Z 482.936,A -85,B 0,C 180,E1 -19859.436,E2 -19859.436} C_VEL
LIN {X 0,Y 245.829,Z 494.501,A -85,B 0,C 180,E1 -19860.923,E2 -19860.923} C_VEL
LIN {X 0,Y 242.726,Z 504.928,A -85,B 0,C 180,E1 -19862.637,E2 -19862.637} C_VEL
LIN {X 0,Y 239.836,Z 513.474,A -85,B 0,C 180,E1 -19864.393,E2 -19864.393} C_VEL
LIN {X 0,Y 236.897,Z 521.372,A -85,B 0,C 180,E1 -19866.392,E2 -19866.392} C_VEL
LIN {X 0,Y 234.025,Z 529.125,A -85,B 0,C 180,E1 -19868.879,E2 -19868.879} C_VEL
LIN {X 0,Y 231.595,Z 535.355,A -85,B 0,C 180,E1 -19871.421,E2 -19871.421} C_VEL
LIN {X 0,Y 229.429,Z 540.34,A -85,B 0,C 180,E1 -19873.998,E2 -19873.998} C_VEL
LIN {X 0,Y 227.836,Z 544.219,A -85,B 0,C 180,E1 -19876.625,E2 -19876.625} C_VEL
LIN {X 0,Y 226.709,Z 547.098,A -85,B 0,C 180,E1 -19879.282,E2 -19879.282} C_VEL
LIN {X 0,Y 225.836,Z 549.462,A -85,B 0,C 180,E1 -19882.851,E2 -19882.851} C_VEL
LIN {X 0,Y 225.587,Z 550.205,A -85,B 0,C 180,E1 -19885.521,E2 -19885.521} C_VEL
LIN {X 0,Y 225.657,Z 550.073,A -85,B 0,C 180,E1 -19888.217,E2 -19888.217} C_VEL
LIN {X 0,Y 225.756,Z 549.478,A -85,B 0,C 180,E1 -19890.002,E2 -19890.002} C_VEL
LIN {X 0,Y 225.691,Z 548.483,A -85,B 0,C 180,E1 -19891.786,E2 -19891.786} C_VEL
LIN {X 0,Y 225.672,Z 545.893,A -85,B 0,C 180,E1 -19894.747,E2 -19894.747} C_VEL
LIN {X 0,Y 225.832,Z 542.858,A -85,B 0,C 180,E1 -19897.152,E2 -19897.152} C_VEL
LIN {X 0,Y 226.263,Z 538.446,A -85,B 0,C 180,E1 -19899.838,E2 -19899.838} C_VEL
LIN {X 0,Y 227.008,Z 532.809,A -85,B 0,C 180,E1 -19902.518,E2 -19902.518} C_VEL
LIN {X 0,Y 228.243,Z 525.752,A -85,B 0,C 180,E1 -19905.174,E2 -19905.174} C_VEL
LIN {X 0,Y 229.596,Z 518.533,A -85,B 0,C 180,E1 -19907.366,E2 -19907.366} C_VEL
LIN {X 0,Y 231.081,Z 509.743,A -85,B 0,C 180,E1 -19909.547,E2 -19909.547} C_VEL
LIN {X 0,Y 232.959,Z 498.915,A -85,B 0,C 180,E1 -19911.69,E2 -19911.69} C_VEL
LIN {X 0,Y 234.726,Z 488.122,A -85,B 0,C 180,E1 -19913.375,E2 -19913.375} C_VEL
LIN {X 0,Y 236.576,Z 476.021,A -85,B 0,C 180,E1 -19914.812,E2 -19914.812} C_VEL
LIN {X 0,Y 238.003,Z 463.351,A -85,B 0,C 180,E1 -19915.939,E2 -19915.939} C_VEL
LIN {X 0,Y 239.077,Z 451.077,A -85,B 0,C 180,E1 -19916.695,E2 -19916.695} C_VEL
LIN {X 0,Y 239.818,Z 435.492,A -85,B 0,C 180,E1 -19917.253,E2 -19917.253} C_VEL
LIN {X 0,Y 241.237,Z 387.884,A -85,B 0,C 180,E1 -19918.641,E2 -19918.641} C_VEL
LIN {X 0,Y 237.451,Z 357.524,A -85,B 0,C 180,E1 -19920.033,E2 -19920.033} C_VEL
LIN {X 0,Y 231.271,Z 340.628,A -85,B 0,C 180,E1 -19921.313,E2 -19921.313} C_VEL
LIN {X 0,Y 230.238,Z 337.713,A -85,B 0,C 180,E1 -19921.572,E2 -19921.572} C_VEL
LIN {X 0,Y 227.894,Z 327.095,A -85,B 0,C 180,E1 -19926.074,E2 -19926.074} C_VEL
LIN {X 0,Y 227.803,Z 327.113,A -85,B 0,C 180,E1 -19930.383,E2 -19930.383} C_VEL
LIN {X 0,Y 227.827,Z 327.108,A -85,B 0,C 180,E1 -19935.196,E2 -19935.196} C_VEL
LIN {X 0,Y 227.83,Z 327.106,A -85,B 0,C 180,E1 -19939.624,E2 -19939.624} C_VEL
LIN {X 0,Y 227.885,Z 327.098,A -85,B 0,C 180,E1 -19944.129,E2 -19944.129} C_VEL
LIN {X 0,Y 227.862,Z 327.1,A -85,B 0,C 180,E1 -19948.376,E2 -19948.376} C_VEL
LIN {X 0,Y 227.862,Z 327.099,A -85,B 0,C 180,E1 -19952.441,E2 -19952.441} C_VEL
LIN {X 0,Y 227.903,Z 327.094,A -85,B 0,C 180,E1 -19956.366,E2 -19956.366} C_VEL
LIN {X 0,Y 227.925,Z 327.076,A -85,B 0,C 180,E1 -19960.173,E2 -19960.173} C_VEL
LIN {X 0,Y 228.026,Z 327.08,A -85,B 0,C 180,E1 -19963.895,E2 -19963.895} C_VEL
LIN {X 0,Y 228.07,Z 327.07,A -85,B 0,C 180,E1 -19967.543,E2 -19967.543} C_VEL
LIN {X 0,Y 228.266,Z 327.028,A -85,B 0,C 180,E1 -19971.144,E2 -19971.144} C_VEL
LIN {X 0,Y 228.318,Z 327.033,A -85,B 0,C 180,E1 -19972.927,E2 -19972.927} C_VEL
LIN {X 0,Y 228.545,Z 327.012,A -85,B 0,C 180,E1 -19978.237,E2 -19978.237} C_VEL
LIN {X 0,Y 228.546,Z 326.995,A -85,B 0,C 180,E1 -19981.762,E2 -19981.762} C_VEL
LIN {X 0,Y 228.312,Z 327.042,A -85,B 0,C 180,E1 -19987.072,E2 -19987.072} C_VEL
LIN {X 0,Y 228.149,Z 327.062,A -85,B 0,C 180,E1 -19990.651,E2 -19990.651} C_VEL
LIN {X 0,Y 228.045,Z 327.057,A -85,B 0,C 180,E1 -19994.273,E2 -19994.273} C_VEL
LIN {X 0,Y 227.94,Z 327.08,A -85,B 0,C 180,E1 -19997.958,E2 -19997.958} C_VEL
LIN {X 0,Y 227.924,Z 327.091,A -85,B 0,C 180,E1 -20002.322,E2 -20002.322} C_VEL
LIN {X 0,Y 227.926,Z 327.074,A -85,B 0,C 180,E1 -20006.591,E2 -20006.591} C_VEL
LIN {X 0,Y 227.877,Z 327.088,A -85,B 0,C 180,E1 -20010.28,E2 -20010.28} C_VEL
LIN {X 0,Y 227.88,Z 327.096,A -85,B 0,C 180,E1 -20013.72,E2 -20013.72} C_VEL
LIN {X 0,Y 227.846,Z 327.081,A -85,B 0,C 180,E1 -20018.09,E2 -20018.09} C_VEL
LIN {X 0,Y 227.813,Z 327.104,A -85,B 0,C 180,E1 -20022.741,E2 -20022.741} C_VEL
LIN {X 0,Y 227.809,Z 327.094,A -85,B 0,C 180,E1 -20027.255,E2 -20027.255} C_VEL
LIN {X 0,Y 227.845,Z 327.105,A -85,B 0,C 180,E1 -20031.908,E2 -20031.908} C_VEL
LIN {X 0,Y 227.881,Z 327.093,A -85,B 0,C 180,E1 -20036.376,E2 -20036.376} C_VEL
LIN {X 0,Y 227.88,Z 327.101,A -85,B 0,C 180,E1 -20040.431,E2 -20040.431} C_VEL
LIN {X 0,Y 227.907,Z 327.097,A -85,B 0,C 180,E1 -20044.422,E2 -20044.422} C_VEL
LIN {X 0,Y 227.957,Z 327.091,A -85,B 0,C 180,E1 -20048.285,E2 -20048.285} C_VEL
LIN {X 0,Y 227.988,Z 327.087,A -85,B 0,C 180,E1 -20052.259,E2 -20052.259} C_VEL
LIN {X 0,Y 229.125,Z 330.113,A -85,B 0,C 180,E1 -20052.523,E2 -20052.523} C_VEL
LIN {X 0,Y 233.098,Z 338.691,A -85,B 0,C 180,E1 -20053.3,E2 -20053.3} C_VEL
LIN {X 0,Y 239.727,Z 356.693,A -85,B 0,C 180,E1 -20054.651,E2 -20054.651} C_VEL
LIN {X 0,Y 241.598,Z 362.823,A -85,B 0,C 180,E1 -20055.051,E2 -20055.051} C_VEL
LIN {X 0,Y 241.99,Z 365.973,A -85,B 0,C 180,E1 -20055.194,E2 -20055.194} C_VEL
LIN {X 0,Y 239.533,Z 433.998,A -85,B 0,C 180,E1 -20057.179,E2 -20057.179} C_VEL
LIN {X 0,Y 238.567,Z 447.183,A -85,B 0,C 180,E1 -20057.882,E2 -20057.882} C_VEL
LIN {X 0,Y 237.387,Z 459.827,A -85,B 0,C 180,E1 -20058.904,E2 -20058.904} C_VEL
LIN {X 0,Y 236.082,Z 471.08,A -85,B 0,C 180,E1 -20060.142,E2 -20060.142} C_VEL
LIN {X 0,Y 234.326,Z 482.62,A -85,B 0,C 180,E1 -20061.787,E2 -20061.787} C_VEL
LIN {X 0,Y 232.449,Z 493.253,A -85,B 0,C 180,E1 -20063.706,E2 -20063.706} C_VEL
LIN {X 0,Y 230.918,Z 501.819,A -85,B 0,C 180,E1 -20065.635,E2 -20065.635} C_VEL
LIN {X 0,Y 229.448,Z 509.718,A -85,B 0,C 180,E1 -20067.804,E2 -20067.804} C_VEL
LIN {X 0,Y 228.008,Z 517.429,A -85,B 0,C 180,E1 -20070.44,E2 -20070.44} C_VEL
LIN {X 0,Y 226.777,Z 524.537,A -85,B 0,C 180,E1 -20073.552,E2 -20073.552} C_VEL
LIN {X 0,Y 226.224,Z 529.207,A -85,B 0,C 180,E1 -20076.214,E2 -20076.214} C_VEL
LIN {X 0,Y 225.701,Z 532.865,A -85,B 0,C 180,E1 -20078.955,E2 -20078.955} C_VEL
LIN {X 0,Y 225.455,Z 534.706,A -85,B 0,C 180,E1 -20080.778,E2 -20080.778} C_VEL
LIN {X 0,Y 225.391,Z 536.089,A -85,B 0,C 180,E1 -20082.606,E2 -20082.606} C_VEL
LIN {X 0,Y 225.416,Z 537.257,A -85,B 0,C 180,E1 -20084.87,E2 -20084.87} C_VEL
LIN {X 0,Y 225.65,Z 537.772,A -85,B 0,C 180,E1 -20088.145,E2 -20088.145} C_VEL
LIN {X 0,Y 226.379,Z 537.008,A -85,B 0,C 180,E1 -20091.354,E2 -20091.354} C_VEL
LIN {X 0,Y 227.108,Z 535.646,A -85,B 0,C 180,E1 -20093.72,E2 -20093.72} C_VEL
LIN {X 0,Y 228.659,Z 532.533,A -85,B 0,C 180,E1 -20096.959,E2 -20096.959} C_VEL
LIN {X 0,Y 230.789,Z 527.953,A -85,B 0,C 180,E1 -20100.161,E2 -20100.161} C_VEL
LIN {X 0,Y 233.133,Z 522.664,A -85,B 0,C 180,E1 -20102.86,E2 -20102.86} C_VEL
LIN {X 0,Y 235.895,Z 515.897,A -85,B 0,C 180,E1 -20105.516,E2 -20105.516} C_VEL
LIN {X 0,Y 239.097,Z 507.399,A -85,B 0,C 180,E1 -20108.115,E2 -20108.115} C_VEL
LIN {X 0,Y 242.21,Z 498.627,A -85,B 0,C 180,E1 -20110.209,E2 -20110.209} C_VEL
LIN {X 0,Y 245.469,Z 488.142,A -85,B 0,C 180,E1 -20112.172,E2 -20112.172} C_VEL
LIN {X 0,Y 248.464,Z 476.657,A -85,B 0,C 180,E1 -20113.866,E2 -20113.866} C_VEL
LIN {X 0,Y 250.969,Z 465.433,A -85,B 0,C 180,E1 -20115.119,E2 -20115.119} C_VEL
LIN {X 0,Y 253.103,Z 452.466,A -85,B 0,C 180,E1 -20116.213,E2 -20116.213} C_VEL
LIN {X 0,Y 254.661,Z 439.419,A -85,B 0,C 180,E1 -20116.972,E2 -20116.972} C_VEL
LIN {X 0,Y 255.668,Z 424.785,A -85,B 0,C 180,E1 -20117.464,E2 -20117.464} C_VEL
LIN {X 0,Y 257.969,Z 380.079,A -85,B 0,C 180,E1 -20118.651,E2 -20118.651} C_VEL
LIN {X 0,Y 251.302,Z 365.824,A -85,B 0,C 180,E1 -20120.489,E2 -20120.489} C_VEL
LIN {X 0,Y 244.7,Z 353.794,A -85,B 0,C 180,E1 -20122.388,E2 -20122.388} C_VEL
LIN {X 0,Y 239.319,Z 344.809,A -85,B 0,C 180,E1 -20124.032,E2 -20124.032} C_VEL
LIN {X 0,Y 234.329,Z 337.123,A -85,B 0,C 180,E1 -20125.652,E2 -20125.652} C_VEL
LIN {X 0,Y 230.546,Z 331.751,A -85,B 0,C 180,E1 -20126.942,E2 -20126.942} C_VEL
LIN {X 0,Y 228.661,Z 329.534,A -85,B 0,C 180,E1 -20127.592,E2 -20127.592} C_VEL
LIN {X 0,Y 228.005,Z 327.807,A -85,B 0,C 180,E1 -20127.879,E2 -20127.879} C_VEL
LIN {X 0,Y 227.849,Z 327.094,A -85,B 0,C 180,E1 -20128.375,E2 -20128.375} C_VEL
LIN {X 0,Y 227.847,Z 327.105,A -85,B 0,C 180,E1 -20132.44,E2 -20132.44} C_VEL
LIN {X 0,Y 227.881,Z 327.099,A -85,B 0,C 180,E1 -20136.364,E2 -20136.364} C_VEL
LIN {X 0,Y 227.882,Z 327.099,A -85,B 0,C 180,E1 -20140.169,E2 -20140.169} C_VEL
LIN {X 0,Y 228,Z 327.082,A -85,B 0,C 180,E1 -20143.894,E2 -20143.894} C_VEL
LIN {X 0,Y 228.116,Z 327.068,A -85,B 0,C 180,E1 -20149.348,E2 -20149.348} C_VEL
LIN {X 0,Y 228.289,Z 327.038,A -85,B 0,C 180,E1 -20152.927,E2 -20152.927} C_VEL
LIN {X 0,Y 228.49,Z 327.014,A -85,B 0,C 180,E1 -20158.238,E2 -20158.238} C_VEL
LIN {X 0,Y 228.525,Z 327.001,A -85,B 0,C 180,E1 -20161.763,E2 -20161.763} C_VEL
LIN {X 0,Y 228.294,Z 327.029,A -85,B 0,C 180,E1 -20167.074,E2 -20167.074} C_VEL
LIN {X 0,Y 228.135,Z 327.066,A -85,B 0,C 180,E1 -20170.652,E2 -20170.652} C_VEL
LIN {X 0,Y 228.033,Z 327.064,A -85,B 0,C 180,E1 -20174.275,E2 -20174.275} C_VEL
LIN {X 0,Y 227.963,Z 327.069,A -85,B 0,C 180,E1 -20177.957,E2 -20177.957} C_VEL
LIN {X 0,Y 227.905,Z 327.082,A -85,B 0,C 180,E1 -20182.319,E2 -20182.319} C_VEL
LIN {X 0,Y 227.9,Z 327.088,A -85,B 0,C 180,E1 -20186.585,E2 -20186.585} C_VEL
LIN {X 0,Y 227.82,Z 327.094,A -85,B 0,C 180,E1 -20188.193,E2 -20188.193} C_VEL
LIN {X 0,Y 227.143,Z 327.193,A -85,B 0,C 180,E1 -20189.669,E2 -20189.669} C_VEL
LIN {X 0,Y 224.277,Z 327.538,A -85,B 0,C 180,E1 -20192.078,E2 -20192.078} C_VEL
LIN {X 0,Y 221.856,Z 327.849,A -85,B 0,C 180,E1 -20194.043,E2 -20194.043} C_VEL
LIN {X 0,Y 220.834,Z 327.968,A -85,B 0,C 180,E1 -20195.569,E2 -20195.569} C_VEL
LIN {X 0,Y 220.76,Z 327.977,A -85,B 0,C 180,E1 -20196.086,E2 -20196.086} C_VEL
LIN {X 0,Y 220.784,Z 328.039,A -85,B 0,C 180,E1 -20199.394,E2 -20199.394} C_VEL
LIN {X 0,Y 223.175,Z 335.771,A -85,B 0,C 180,E1 -20204.64,E2 -20204.64} C_VEL
LIN {X 0,Y 226.249,Z 340.751,A -85,B 0,C 180,E1 -20205.901,E2 -20205.901} C_VEL
LIN {X 0,Y 227.917,Z 343.413,A -85,B 0,C 180,E1 -20206.52,E2 -20206.52} C_VEL
LIN {X 0,Y 231.276,Z 348.649,A -85,B 0,C 180,E1 -20207.711,E2 -20207.711} C_VEL
LIN {X 0,Y 236.445,Z 357.293,A -85,B 0,C 180,E1 -20209.455,E2 -20209.455} C_VEL
LIN {X 0,Y 242.947,Z 369.699,A -85,B 0,C 180,E1 -20211.525,E2 -20211.525} C_VEL
LIN {X 0,Y 249.145,Z 383.118,A -85,B 0,C 180,E1 -20213.393,E2 -20213.393} C_VEL
LIN {X 0,Y 250.45,Z 386.571,A -85,B 0,C 180,E1 -20213.791,E2 -20213.791} C_VEL
LIN {X 0,Y 251.83,Z 395.418,A -85,B 0,C 180,E1 -20214.399,E2 -20214.399} C_VEL
LIN {X 0,Y 249.185,Z 446.248,A -85,B 0,C 180,E1 -20215.847,E2 -20215.847} C_VEL
LIN {X 0,Y 247.597,Z 459.827,A -85,B 0,C 180,E1 -20216.516,E2 -20216.516} C_VEL
LIN {X 0,Y 245.371,Z 472.139,A -85,B 0,C 180,E1 -20217.398,E2 -20217.398} C_VEL
LIN {X 0,Y 242.735,Z 483.929,A -85,B 0,C 180,E1 -20218.592,E2 -20218.592} C_VEL
LIN {X 0,Y 239.673,Z 495.273,A -85,B 0,C 180,E1 -20220.102,E2 -20220.102} C_VEL
LIN {X 0,Y 236.481,Z 505.526,A -85,B 0,C 180,E1 -20221.851,E2 -20221.851} C_VEL
LIN {X 0,Y 233.485,Z 513.934,A -85,B 0,C 180,E1 -20223.644,E2 -20223.644} C_VEL
LIN {X 0,Y 229.861,Z 523.077,A -85,B 0,C 180,E1 -20226.103,E2 -20226.103} C_VEL
LIN {X 0,Y 226.954,Z 530.445,A -85,B 0,C 180,E1 -20228.665,E2 -20228.665} C_VEL
LIN {X 0,Y 224.055,Z 537.279,A -85,B 0,C 180,E1 -20231.721,E2 -20231.721} C_VEL
LIN {X 0,Y 221.95,Z 541.813,A -85,B 0,C 180,E1 -20234.388,E2 -20234.388} C_VEL
LIN {X 0,Y 220.471,Z 545.281,A -85,B 0,C 180,E1 -20237.108,E2 -20237.108} C_VEL
LIN {X 0,Y 219.166,Z 548.376,A -85,B 0,C 180,E1 -20240.775,E2 -20240.775} C_VEL
LIN {X 0,Y 218.571,Z 549.914,A -85,B 0,C 180,E1 -20244.466,E2 -20244.466} C_VEL
LIN {X 0,Y 218.499,Z 550.069,A -85,B 0,C 180,E1 -20246.313,E2 -20246.313} C_VEL
LIN {X 0,Y 218.572,Z 549.831,A -85,B 0,C 180,E1 -20248.159,E2 -20248.159} C_VEL
LIN {X 0,Y 218.668,Z 549.206,A -85,B 0,C 180,E1 -20250.002,E2 -20250.002} C_VEL
LIN {X 0,Y 218.606,Z 548.182,A -85,B 0,C 180,E1 -20251.844,E2 -20251.844} C_VEL
LIN {X 0,Y 218.577,Z 545.813,A -85,B 0,C 180,E1 -20254.611,E2 -20254.611} C_VEL
LIN {X 0,Y 218.784,Z 542.432,A -85,B 0,C 180,E1 -20257.384,E2 -20257.384} C_VEL
LIN {X 0,Y 219.253,Z 537.95,A -85,B 0,C 180,E1 -20260.156,E2 -20260.156} C_VEL
LIN {X 0,Y 220.024,Z 532.235,A -85,B 0,C 180,E1 -20262.922,E2 -20262.922} C_VEL
LIN {X 0,Y 221.367,Z 525.056,A -85,B 0,C 180,E1 -20265.657,E2 -20265.657} C_VEL
LIN {X 0,Y 222.814,Z 517.737,A -85,B 0,C 180,E1 -20267.912,E2 -20267.912} C_VEL
LIN {X 0,Y 224.335,Z 508.819,A -85,B 0,C 180,E1 -20270.16,E2 -20270.16} C_VEL
LIN {X 0,Y 226.11,Z 499.036,A -85,B 0,C 180,E1 -20272.142,E2 -20272.142} C_VEL
LIN {X 0,Y 227.931,Z 488.322,A -85,B 0,C 180,E1 -20273.874,E2 -20273.874} C_VEL
LIN {X 0,Y 229.833,Z 476.36,A -85,B 0,C 180,E1 -20275.349,E2 -20275.349} C_VEL
LIN {X 0,Y 231.314,Z 463.856,A -85,B 0,C 180,E1 -20276.505,E2 -20276.505} C_VEL
LIN {X 0,Y 232.488,Z 451.064,A -85,B 0,C 180,E1 -20277.325,E2 -20277.325} C_VEL
LIN {X 0,Y 233.245,Z 435.964,A -85,B 0,C 180,E1 -20277.886,E2 -20277.886} C_VEL
LIN {X 0,Y 234.719,Z 388.675,A -85,B 0,C 180,E1 -20279.3,E2 -20279.3} C_VEL
LIN {X 0,Y 231.16,Z 359.609,A -85,B 0,C 180,E1 -20280.679,E2 -20280.679} C_VEL
LIN {X 0,Y 225.465,Z 343.929,A -85,B 0,C 180,E1 -20281.913,E2 -20281.913} C_VEL
LIN {X 0,Y 222.944,Z 337.547,A -85,B 0,C 180,E1 -20282.48,E2 -20282.48} C_VEL
LIN {X 0,Y 220.83,Z 327.979,A -85,B 0,C 180,E1 -20286.709,E2 -20286.709} C_VEL
LIN {X 0,Y 220.775,Z 327.989,A -85,B 0,C 180,E1 -20290.181,E2 -20290.181} C_VEL
LIN {X 0,Y 220.766,Z 327.991,A -85,B 0,C 180,E1 -20294.458,E2 -20294.458} C_VEL
LIN {X 0,Y 220.772,Z 327.988,A -85,B 0,C 180,E1 -20298.047,E2 -20298.047} C_VEL
LIN {X 0,Y 220.812,Z 327.983,A -85,B 0,C 180,E1 -20300.464,E2 -20300.464} C_VEL
LIN {X 0,Y 220.806,Z 327.979,A -85,B 0,C 180,E1 -20305.045,E2 -20305.045} C_VEL
LIN {X 0,Y 220.84,Z 327.975,A -85,B 0,C 180,E1 -20309.39,E2 -20309.39} C_VEL
LIN {X 0,Y 220.882,Z 327.97,A -85,B 0,C 180,E1 -20313.547,E2 -20313.547} C_VEL
LIN {X 0,Y 220.873,Z 327.965,A -85,B 0,C 180,E1 -20317.552,E2 -20317.552} C_VEL
LIN {X 0,Y 220.934,Z 327.957,A -85,B 0,C 180,E1 -20322.618,E2 -20322.618} C_VEL
LIN {X 0,Y 221.007,Z 327.953,A -85,B 0,C 180,E1 -20327.138,E2 -20327.138} C_VEL
LIN {X 0,Y 221.204,Z 327.906,A -85,B 0,C 180,E1 -20330.859,E2 -20330.859} C_VEL
LIN {X 0,Y 221.254,Z 327.913,A -85,B 0,C 180,E1 -20332.7,E2 -20332.7} C_VEL
LIN {X 0,Y 221.479,Z 327.892,A -85,B 0,C 180,E1 -20338.181,E2 -20338.181} C_VEL
LIN {X 0,Y 221.58,Z 327.871,A -85,B 0,C 180,E1 -20340,E2 -20340} C_VEL
LIN {X 0,Y 221.48,Z 327.873,A -85,B 0,C 180,E1 -20341.818,E2 -20341.818} C_VEL
LIN {X 0,Y 221.249,Z 327.921,A -85,B 0,C 180,E1 -20347.299,E2 -20347.299} C_VEL
LIN {X 0,Y 221.07,Z 327.941,A -85,B 0,C 180,E1 -20350.996,E2 -20350.996} C_VEL
LIN {X 0,Y 220.973,Z 327.934,A -85,B 0,C 180,E1 -20354.74,E2 -20354.74} C_VEL
LIN {X 0,Y 220.884,Z 327.961,A -85,B 0,C 180,E1 -20358.552,E2 -20358.552} C_VEL
LIN {X 0,Y 220.872,Z 327.972,A -85,B 0,C 180,E1 -20362.663,E2 -20362.663} C_VEL
LIN {X 0,Y 220.869,Z 327.949,A -85,B 0,C 180,E1 -20367.004,E2 -20367.004} C_VEL
LIN {X 0,Y 220.822,Z 327.968,A -85,B 0,C 180,E1 -20370.758,E2 -20370.758} C_VEL
LIN {X 0,Y 220.804,Z 327.976,A -85,B 0,C 180,E1 -20374.954,E2 -20374.954} C_VEL
LIN {X 0,Y 220.81,Z 327.96,A -85,B 0,C 180,E1 -20379.536,E2 -20379.536} C_VEL
LIN {X 0,Y 220.774,Z 327.98,A -85,B 0,C 180,E1 -20384.453,E2 -20384.453} C_VEL
LIN {X 0,Y 220.77,Z 327.97,A -85,B 0,C 180,E1 -20388.046,E2 -20388.046} C_VEL
LIN {X 0,Y 220.809,Z 327.98,A -85,B 0,C 180,E1 -20390.462,E2 -20390.462} C_VEL
LIN {X 0,Y 220.803,Z 327.968,A -85,B 0,C 180,E1 -20395.044,E2 -20395.044} C_VEL
LIN {X 0,Y 220.836,Z 327.974,A -85,B 0,C 180,E1 -20399.388,E2 -20399.388} C_VEL
LIN {X 0,Y 220.879,Z 327.97,A -85,B 0,C 180,E1 -20403.546,E2 -20403.546} C_VEL
LIN {X 0,Y 220.872,Z 327.973,A -85,B 0,C 180,E1 -20407.551,E2 -20407.551} C_VEL
LIN {X 0,Y 220.913,Z 328.032,A -85,B 0,C 180,E1 -20411.388,E2 -20411.388} C_VEL
LIN {X 0,Y 222.004,Z 330.945,A -85,B 0,C 180,E1 -20411.639,E2 -20411.639} C_VEL
LIN {X 0,Y 226.487,Z 340.06,A -85,B 0,C 180,E1 -20412.542,E2 -20412.542} C_VEL
LIN {X 0,Y 233.33,Z 358.411,A -85,B 0,C 180,E1 -20413.994,E2 -20413.994} C_VEL
LIN {X 0,Y 235.37,Z 365.259,A -85,B 0,C 180,E1 -20414.454,E2 -20414.454} C_VEL
LIN {X 0,Y 233.91,Z 410.712,A -85,B 0,C 180,E1 -20415.808,E2 -20415.808} C_VEL
LIN {X 0,Y 232.866,Z 435.322,A -85,B 0,C 180,E1 -20416.583,E2 -20416.583} C_VEL
LIN {X 0,Y 231.852,Z 448.867,A -85,B 0,C 180,E1 -20417.359,E2 -20417.359} C_VEL
LIN {X 0,Y 230.552,Z 461.58,A -85,B 0,C 180,E1 -20418.459,E2 -20418.459} C_VEL
LIN {X 0,Y 229.154,Z 473.006,A -85,B 0,C 180,E1 -20419.809,E2 -20419.809} C_VEL
LIN {X 0,Y 227.205,Z 484.939,A -85,B 0,C 180,E1 -20421.616,E2 -20421.616} C_VEL
LIN {X 0,Y 225.26,Z 495.712,A -85,B 0,C 180,E1 -20423.729,E2 -20423.729} C_VEL
LIN {X 0,Y 223.469,Z 504.723,A -85,B 0,C 180,E1 -20425.941,E2 -20425.941} C_VEL
LIN {X 0,Y 221.743,Z 513.512,A -85,B 0,C 180,E1 -20428.636,E2 -20428.636} C_VEL
LIN {X 0,Y 220.479,Z 520.508,A -85,B 0,C 180,E1 -20431.368,E2 -20431.368} C_VEL
LIN {X 0,Y 219.479,Z 526.924,A -85,B 0,C 180,E1 -20434.59,E2 -20434.59} C_VEL
LIN {X 0,Y 218.867,Z 531.15,A -85,B 0,C 180,E1 -20437.378,E2 -20437.378} C_VEL
LIN {X 0,Y 218.54,Z 533.392,A -85,B 0,C 180,E1 -20439.251,E2 -20439.251} C_VEL
LIN {X 0,Y 218.325,Z 535.139,A -85,B 0,C 180,E1 -20441.134,E2 -20441.134} C_VEL
LIN {X 0,Y 218.274,Z 536.471,A -85,B 0,C 180,E1 -20443.024,E2 -20443.024} C_VEL
LIN {X 0,Y 218.338,Z 537.455,A -85,B 0,C 180,E1 -20445.061,E2 -20445.061} C_VEL
LIN {X 0,Y 218.639,Z 537.951,A -85,B 0,C 180,E1 -20448.748,E2 -20448.748} C_VEL
LIN {X 0,Y 219.372,Z 537.231,A -85,B 0,C 180,E1 -20451.71,E2 -20451.71} C_VEL
LIN {X 0,Y 220.311,Z 535.615,A -85,B 0,C 180,E1 -20454.499,E2 -20454.499} C_VEL
LIN {X 0,Y 221.804,Z 532.803,A -85,B 0,C 180,E1 -20457.477,E2 -20457.477} C_VEL
LIN {X 0,Y 223.619,Z 529.163,A -85,B 0,C 180,E1 -20460.187,E2 -20460.187} C_VEL
LIN {X 0,Y 226.194,Z 523.71,A -85,B 0,C 180,E1 -20463.195,E2 -20463.195} C_VEL
LIN {X 0,Y 228.809,Z 517.795,A -85,B 0,C 180,E1 -20465.702,E2 -20465.702} C_VEL
LIN {X 0,Y 232.016,Z 509.841,A -85,B 0,C 180,E1 -20468.346,E2 -20468.346} C_VEL
LIN {X 0,Y 235.239,Z 501.415,A -85,B 0,C 180,E1 -20470.524,E2 -20470.524} C_VEL
LIN {X 0,Y 238.678,Z 491.172,A -85,B 0,C 180,E1 -20472.626,E2 -20472.626} C_VEL
LIN {X 0,Y 241.632,Z 480.991,A -85,B 0,C 180,E1 -20474.269,E2 -20474.269} C_VEL
LIN {X 0,Y 244.37,Z 469.782,A -85,B 0,C 180,E1 -20475.673,E2 -20475.673} C_VEL
LIN {X 0,Y 246.682,Z 458.072,A -85,B 0,C 180,E1 -20476.793,E2 -20476.793} C_VEL
LIN {X 0,Y 248.545,Z 445.037,A -85,B 0,C 180,E1 -20477.705,E2 -20477.705} C_VEL
LIN {X 0,Y 249.726,Z 432.156,A -85,B 0,C 180,E1 -20478.277,E2 -20478.277} C_VEL
LIN {X 0,Y 252.388,Z 382.12,A -85,B 0,C 180,E1 -20479.653,E2 -20479.653} C_VEL
LIN {X 0,Y 246.104,Z 368.827,A -85,B 0,C 180,E1 -20481.472,E2 -20481.472} C_VEL
LIN {X 0,Y 240.578,Z 358.603,A -85,B 0,C 180,E1 -20483.146,E2 -20483.146} C_VEL
LIN {X 0,Y 234.011,Z 347.424,A -85,B 0,C 180,E1 -20485.272,E2 -20485.272} C_VEL
LIN {X 0,Y 229.24,Z 340.343,A -85,B 0,C 180,E1 -20486.909,E2 -20486.909} C_VEL
LIN {X 0,Y 227.331,Z 337.608,A -85,B 0,C 180,E1 -20487.594,E2 -20487.594} C_VEL
LIN {X 0,Y 224.981,Z 334.564,A -85,B 0,C 180,E1 -20488.451,E2 -20488.451} C_VEL
LIN {X 0,Y 224.277,Z 333.235,A -85,B 0,C 180,E1 -20488.735,E2 -20488.735} C_VEL
LIN {X 0,Y 221.999,Z 331.107,A -85,B 0,C 180,E1 -20489.568,E2 -20489.568} C_VEL
LIN {X 0,Y 221.004,Z 328.927,A -85,B 0,C 180,E1 -20490.01,E2 -20490.01} C_VEL
LIN {X 0,Y 220.822,Z 327.989,A -85,B 0,C 180,E1 -20490.212,E2 -20490.212} C_VEL
LIN {X 0,Y 220.868,Z 327.965,A -85,B 0,C 180,E1 -20493.546,E2 -20493.546} C_VEL
LIN {X 0,Y 220.846,Z 327.965,A -85,B 0,C 180,E1 -20497.55,E2 -20497.55} C_VEL
LIN {X 0,Y 220.907,Z 327.955,A -85,B 0,C 180,E1 -20502.629,E2 -20502.629} C_VEL
LIN {X 0,Y 220.955,Z 327.946,A -85,B 0,C 180,E1 -20507.136,E2 -20507.136} C_VEL
LIN {X 0,Y 221.178,Z 327.917,A -85,B 0,C 180,E1 -20510.859,E2 -20510.859} C_VEL
LIN {X 0,Y 221.226,Z 327.915,A -85,B 0,C 180,E1 -20512.7,E2 -20512.7} C_VEL
LIN {X 0,Y 221.427,Z 327.892,A -85,B 0,C 180,E1 -20518.182,E2 -20518.182} C_VEL
LIN {X 0,Y 221.532,Z 327.889,A -85,B 0,C 180,E1 -20520,E2 -20520} C_VEL
LIN {X 0,Y 221.458,Z 327.881,A -85,B 0,C 180,E1 -20521.819,E2 -20521.819} C_VEL
LIN {X 0,Y 221.232,Z 327.907,A -85,B 0,C 180,E1 -20527.301,E2 -20527.301} C_VEL
LIN {X 0,Y 221.055,Z 327.944,A -85,B 0,C 180,E1 -20530.997,E2 -20530.997} C_VEL
LIN {X 0,Y 220.984,Z 327.948,A -85,B 0,C 180,E1 -20536.633,E2 -20536.633} C_VEL
LIN {X 0,Y 220.871,Z 327.968,A -85,B 0,C 180,E1 -20540.489,E2 -20540.489} C_VEL
LIN {X 0,Y 220.823,Z 327.969,A -85,B 0,C 180,E1 -20544.441,E2 -20544.441} C_VEL
LIN {X 0,Y 220.794,Z 327.972,A -85,B 0,C 180,E1 -20548.52,E2 -20548.52} C_VEL
LIN {X 0,Y 220.806,Z 327.974,A -85,B 0,C 180,E1 -20552.758,E2 -20552.758} C_VEL
LIN {X 0,Y 220.76,Z 327.977,A -85,B 0,C 180,E1 -20556.086,E2 -20556.086} C_VEL
LIN {X 0,Y 220.189,Z 328.362,A -85,B 0,C 180,E1 -20557.102,E2 -20557.102} C_VEL
LIN {X 0,Y 218.859,Z 329.317,A -85,B 0,C 180,E1 -20558.064,E2 -20558.064} C_VEL
LIN {X 0,Y 215.624,Z 332.682,A -85,B 0,C 180,E1 -20560.257,E2 -20560.257} C_VEL
LIN {X 0,Y 215.388,Z 334.196,A -85,B 0,C 180,E1 -20561.251,E2 -20561.251} C_VEL
LIN {X 0,Y 215.898,Z 335.737,A -85,B 0,C 180,E1 -20562.253,E2 -20562.253} C_VEL
LIN {X 0,Y 218.842,Z 340.347,A -85,B 0,C 180,E1 -20563.533,E2 -20563.533} C_VEL
LIN {X 0,Y 220.444,Z 342.537,A -85,B 0,C 180,E1 -20564.181,E2 -20564.181} C_VEL
LIN {X 0,Y 224.223,Z 348.446,A -85,B 0,C 180,E1 -20565.669,E2 -20565.669} C_VEL
LIN {X 0,Y 227.789,Z 354.206,A -85,B 0,C 180,E1 -20566.997,E2 -20566.997} C_VEL
LIN {X 0,Y 232.63,Z 362.465,A -85,B 0,C 180,E1 -20568.703,E2 -20568.703} C_VEL
LIN {X 0,Y 238.514,Z 373.885,A -85,B 0,C 180,E1 -20570.668,E2 -20570.668} C_VEL
LIN {X 0,Y 244.636,Z 387.473,A -85,B 0,C 180,E1 -20572.613,E2 -20572.613} C_VEL
LIN {X 0,Y 245.495,Z 390.264,A -85,B 0,C 180,E1 -20572.908,E2 -20572.908} C_VEL
LIN {X 0,Y 246.448,Z 396.673,A -85,B 0,C 180,E1 -20573.359,E2 -20573.359} C_VEL
LIN {X 0,Y 243.75,Z 446.088,A -85,B 0,C 180,E1 -20574.786,E2 -20574.786} C_VEL
LIN {X 0,Y 242.228,Z 458.898,A -85,B 0,C 180,E1 -20575.42,E2 -20575.42} C_VEL
LIN {X 0,Y 239.931,Z 471.413,A -85,B 0,C 180,E1 -20576.311,E2 -20576.311} C_VEL
LIN {X 0,Y 237.165,Z 483.352,A -85,B 0,C 180,E1 -20577.515,E2 -20577.515} C_VEL
LIN {X 0,Y 233.991,Z 494.765,A -85,B 0,C 180,E1 -20579.048,E2 -20579.048} C_VEL
LIN {X 0,Y 231.005,Z 504.01,A -85,B 0,C 180,E1 -20580.623,E2 -20580.623} C_VEL
LIN {X 0,Y 227.179,Z 514.377,A -85,B 0,C 180,E1 -20582.853,E2 -20582.853} C_VEL
LIN {X 0,Y 223.412,Z 523.39,A -85,B 0,C 180,E1 -20585.368,E2 -20585.368} C_VEL
LIN {X 0,Y 220.363,Z 530.667,A -85,B 0,C 180,E1 -20587.994,E2 -20587.994} C_VEL
LIN {X 0,Y 217.318,Z 537.383,A -85,B 0,C 180,E1 -20591.133,E2 -20591.133} C_VEL
LIN {X 0,Y 215.107,Z 541.845,A -85,B 0,C 180,E1 -20593.878,E2 -20593.878} C_VEL
LIN {X 0,Y 213.534,Z 545.254,A -85,B 0,C 180,E1 -20596.682,E2 -20596.682} C_VEL
LIN {X 0,Y 212.133,Z 548.279,A -85,B 0,C 180,E1 -20600.467,E2 -20600.467} C_VEL
LIN {X 0,Y 211.495,Z 549.742,A -85,B 0,C 180,E1 -20604.28,E2 -20604.28} C_VEL
LIN {X 0,Y 211.398,Z 549.854,A -85,B 0,C 180,E1 -20606.189,E2 -20606.189} C_VEL
LIN {X 0,Y 211.47,Z 549.587,A -85,B 0,C 180,E1 -20608.097,E2 -20608.097} C_VEL
LIN {X 0,Y 211.583,Z 548.935,A -85,B 0,C 180,E1 -20610.002,E2 -20610.002} C_VEL
LIN {X 0,Y 211.502,Z 547.871,A -85,B 0,C 180,E1 -20611.906,E2 -20611.906} C_VEL
LIN {X 0,Y 211.475,Z 545.763,A -85,B 0,C 180,E1 -20614.434,E2 -20614.434} C_VEL
LIN {X 0,Y 211.706,Z 542.003,A -85,B 0,C 180,E1 -20617.632,E2 -20617.632} C_VEL
LIN {X 0,Y 212.215,Z 537.452,A -85,B 0,C 180,E1 -20620.496,E2 -20620.496} C_VEL
LIN {X 0,Y 213.29,Z 530.518,A -85,B 0,C 180,E1 -20623.823,E2 -20623.823} C_VEL
LIN {X 0,Y 214.755,Z 522.984,A -85,B 0,C 180,E1 -20626.641,E2 -20626.641} C_VEL
LIN {X 0,Y 216.379,Z 515.291,A -85,B 0,C 180,E1 -20628.955,E2 -20628.955} C_VEL
LIN {X 0,Y 217.8,Z 506.905,A -85,B 0,C 180,E1 -20631.039,E2 -20631.039} C_VEL
LIN {X 0,Y 219.76,Z 496.737,A -85,B 0,C 180,E1 -20633.066,E2 -20633.066} C_VEL
LIN {X 0,Y 221.769,Z 485.419,A -85,B 0,C 180,E1 -20634.83,E2 -20634.83} C_VEL
LIN {X 0,Y 223.648,Z 472.673,A -85,B 0,C 180,E1 -20636.353,E2 -20636.353} C_VEL
LIN {X 0,Y 225.063,Z 460.184,A -85,B 0,C 180,E1 -20637.427,E2 -20637.427} C_VEL
LIN {X 0,Y 226.218,Z 446.293,A -85,B 0,C 180,E1 -20638.217,E2 -20638.217} C_VEL
LIN {X 0,Y 228.241,Z 389.335,A -85,B 0,C 180,E1 -20640,E2 -20640} C_VEL
LIN {X 0,Y 224.83,Z 361.436,A -85,B 0,C 180,E1 -20641.375,E2 -20641.375} C_VEL
LIN {X 0,Y 219.277,Z 346.302,A -85,B 0,C 180,E1 -20642.629,E2 -20642.629} C_VEL
LIN {X 0,Y 215.663,Z 337.22,A -85,B 0,C 180,E1 -20643.513,E2 -20643.513} C_VEL
LIN {X 0,Y 213.771,Z 328.858,A -85,B 0,C 180,E1 -20647.416,E2 -20647.416} C_VEL
LIN {X 0,Y 213.702,Z 328.867,A -85,B 0,C 180,E1 -20651.129,E2 -20651.129} C_VEL
LIN {X 0,Y 213.707,Z 328.867,A -85,B 0,C 180,E1 -20653.68,E2 -20653.68} C_VEL
LIN {X 0,Y 213.708,Z 328.868,A -85,B 0,C 180,E1 -20656.346,E2 -20656.346} C_VEL
LIN {X 0,Y 213.722,Z 328.864,A -85,B 0,C 180,E1 -20659.144,E2 -20659.144} C_VEL
LIN {X 0,Y 213.749,Z 328.859,A -85,B 0,C 180,E1 -20663.712,E2 -20663.712} C_VEL
LIN {X 0,Y 213.764,Z 328.856,A -85,B 0,C 180,E1 -20668.261,E2 -20668.261} C_VEL
LIN {X 0,Y 213.795,Z 328.852,A -85,B 0,C 180,E1 -20672.598,E2 -20672.598} C_VEL
LIN {X 0,Y 213.817,Z 328.848,A -85,B 0,C 180,E1 -20676.979,E2 -20676.979} C_VEL
LIN {X 0,Y 213.897,Z 328.834,A -85,B 0,C 180,E1 -20682.799,E2 -20682.799} C_VEL
LIN {X 0,Y 213.946,Z 328.831,A -85,B 0,C 180,E1 -20686.706,E2 -20686.706} C_VEL
LIN {X 0,Y 214.143,Z 328.784,A -85,B 0,C 180,E1 -20690.555,E2 -20690.555} C_VEL
LIN {X 0,Y 214.09,Z 328.813,A -85,B 0,C 180,E1 -20694.348,E2 -20694.348} C_VEL
LIN {X 0,Y 214.415,Z 328.772,A -85,B 0,C 180,E1 -20698.121,E2 -20698.121} C_VEL
LIN {X 0,Y 214.545,Z 328.746,A -85,B 0,C 180,E1 -20700,E2 -20700} C_VEL
LIN {X 0,Y 214.416,Z 328.751,A -85,B 0,C 180,E1 -20701.878,E2 -20701.878} C_VEL
LIN {X 0,Y 214.19,Z 328.801,A -85,B 0,C 180,E1 -20707.541,E2 -20707.541} C_VEL
LIN {X 0,Y 214.001,Z 328.821,A -85,B 0,C 180,E1 -20711.364,E2 -20711.364} C_VEL
LIN {X 0,Y 213.907,Z 328.811,A -85,B 0,C 180,E1 -20715.238,E2 -20715.238} C_VEL
LIN {X 0,Y 213.813,Z 328.847,A -85,B 0,C 180,E1 -20719.189,E2 -20719.189} C_VEL
LIN {X 0,Y 213.807,Z 328.848,A -85,B 0,C 180,E1 -20723.231,E2 -20723.231} C_VEL
LIN {X 0,Y 213.79,Z 328.827,A -85,B 0,C 180,E1 -20727.426,E2 -20727.426} C_VEL
LIN {X 0,Y 213.762,Z 328.854,A -85,B 0,C 180,E1 -20731.738,E2 -20731.738} C_VEL
LIN {X 0,Y 213.747,Z 328.846,A -85,B 0,C 180,E1 -20736.287,E2 -20736.287} C_VEL
LIN {X 0,Y 213.715,Z 328.855,A -85,B 0,C 180,E1 -20741.124,E2 -20741.124} C_VEL
LIN {X 0,Y 213.707,Z 328.864,A -85,B 0,C 180,E1 -20743.678,E2 -20743.678} C_VEL
LIN {X 0,Y 213.706,Z 328.851,A -85,B 0,C 180,E1 -20746.344,E2 -20746.344} C_VEL
LIN {X 0,Y 213.719,Z 328.855,A -85,B 0,C 180,E1 -20749.142,E2 -20749.142} C_VEL
LIN {X 0,Y 213.746,Z 328.854,A -85,B 0,C 180,E1 -20753.71,E2 -20753.71} C_VEL
LIN {X 0,Y 213.761,Z 328.86,A -85,B 0,C 180,E1 -20758.26,E2 -20758.26} C_VEL
LIN {X 0,Y 213.792,Z 328.856,A -85,B 0,C 180,E1 -20762.597,E2 -20762.597} C_VEL
LIN {X 0,Y 213.814,Z 328.853,A -85,B 0,C 180,E1 -20766.977,E2 -20766.977} C_VEL
LIN {X 0,Y 213.87,Z 328.847,A -85,B 0,C 180,E1 -20770.42,E2 -20770.42} C_VEL
LIN {X 0,Y 214.879,Z 331.676,A -85,B 0,C 180,E1 -20770.687,E2 -20770.687} C_VEL
LIN {X 0,Y 220.275,Z 342.39,A -85,B 0,C 180,E1 -20771.824,E2 -20771.824} C_VEL
LIN {X 0,Y 226.677,Z 359.535,A -85,B 0,C 180,E1 -20773.247,E2 -20773.247} C_VEL
LIN {X 0,Y 228.962,Z 366.44,A -85,B 0,C 180,E1 -20773.758,E2 -20773.758} C_VEL
LIN {X 0,Y 226.421,Z 434.336,A -85,B 0,C 180,E1 -20775.85,E2 -20775.85} C_VEL
LIN {X 0,Y 225.383,Z 447.541,A -85,B 0,C 180,E1 -20776.588,E2 -20776.588} C_VEL
LIN {X 0,Y 224.117,Z 460.19,A -85,B 0,C 180,E1 -20777.663,E2 -20777.663} C_VEL
LIN {X 0,Y 222.59,Z 472.243,A -85,B 0,C 180,E1 -20779.078,E2 -20779.078} C_VEL
LIN {X 0,Y 220.683,Z 483.771,A -85,B 0,C 180,E1 -20780.836,E2 -20780.836} C_VEL
LIN {X 0,Y 218.691,Z 494.171,A -85,B 0,C 180,E1 -20782.845,E2 -20782.845} C_VEL
LIN {X 0,Y 217.058,Z 502.645,A -85,B 0,C 180,E1 -20784.89,E2 -20784.89} C_VEL
LIN {X 0,Y 215.183,Z 511.829,A -85,B 0,C 180,E1 -20787.659,E2 -20787.659} C_VEL
LIN {X 0,Y 213.713,Z 519.226,A -85,B 0,C 180,E1 -20790.469,E2 -20790.469} C_VEL
LIN {X 0,Y 212.79,Z 524.241,A -85,B 0,C 180,E1 -20792.838,E2 -20792.838} C_VEL
LIN {X 0,Y 212.032,Z 529.671,A -85,B 0,C 180,E1 -20796.081,E2 -20796.081} C_VEL
LIN {X 0,Y 211.559,Z 532.852,A -85,B 0,C 180,E1 -20798.596,E2 -20798.596} C_VEL
LIN {X 0,Y 211.197,Z 535.573,A -85,B 0,C 180,E1 -20801.515,E2 -20801.515} C_VEL
LIN {X 0,Y 211.168,Z 536.854,A -85,B 0,C 180,E1 -20803.47,E2 -20803.47} C_VEL
LIN {X 0,Y 211.263,Z 537.703,A -85,B 0,C 180,E1 -20805.432,E2 -20805.432} C_VEL
LIN {X 0,Y 211.378,Z 538.117,A -85,B 0,C 180,E1 -20807.41,E2 -20807.41} C_VEL
LIN {X 0,Y 211.658,Z 538.13,A -85,B 0,C 180,E1 -20809.391,E2 -20809.391} C_VEL
LIN {X 0,Y 212.369,Z 537.454,A -85,B 0,C 180,E1 -20812.088,E2 -20812.088} C_VEL
LIN {X 0,Y 213.541,Z 535.586,A -85,B 0,C 180,E1 -20815.329,E2 -20815.329} C_VEL
LIN {X 0,Y 215.007,Z 533.051,A -85,B 0,C 180,E1 -20818.049,E2 -20818.049} C_VEL
LIN {X 0,Y 217.174,Z 528.91,A -85,B 0,C 180,E1 -20821.181,E2 -20821.181} C_VEL
LIN {X 0,Y 219.877,Z 523.544,A -85,B 0,C 180,E1 -20824.156,E2 -20824.156} C_VEL
LIN {X 0,Y 222.782,Z 517.272,A -85,B 0,C 180,E1 -20826.823,E2 -20826.823} C_VEL
LIN {X 0,Y 226.131,Z 509.298,A -85,B 0,C 180,E1 -20829.46,E2 -20829.46} C_VEL
LIN {X 0,Y 229.635,Z 500.483,A -85,B 0,C 180,E1 -20831.73,E2 -20831.73} C_VEL
LIN {X 0,Y 232.711,Z 491.675,A -85,B 0,C 180,E1 -20833.547,E2 -20833.547} C_VEL
LIN {X 0,Y 235.986,Z 480.872,A -85,B 0,C 180,E1 -20835.316,E2 -20835.316} C_VEL
LIN {X 0,Y 238.829,Z 469.58,A -85,B 0,C 180,E1 -20836.743,E2 -20836.743} C_VEL
LIN {X 0,Y 241.171,Z 458.075,A -85,B 0,C 180,E1 -20837.851,E2 -20837.851} C_VEL
LIN {X 0,Y 243.109,Z 444.983,A -85,B 0,C 180,E1 -20838.772,E2 -20838.772} C_VEL
LIN {X 0,Y 244.315,Z 432.341,A -85,B 0,C 180,E1 -20839.336,E2 -20839.336} C_VEL
LIN {X 0,Y 246.995,Z 384.581,A -85,B 0,C 180,E1 -20840.66,E2 -20840.66} C_VEL
LIN {X 0,Y 241.264,Z 372.326,A -85,B 0,C 180,E1 -20842.418,E2 -20842.418} C_VEL
LIN {X 0,Y 234.646,Z 360.001,A -85,B 0,C 180,E1 -20844.547,E2 -20844.547} C_VEL
LIN {X 0,Y 227.75,Z 348.572,A -85,B 0,C 180,E1 -20846.945,E2 -20846.945} C_VEL
LIN {X 0,Y 223.921,Z 343.146,A -85,B 0,C 180,E1 -20848.35,E2 -20848.35} C_VEL
LIN {X 0,Y 220.611,Z 338.774,A -85,B 0,C 180,E1 -20849.624,E2 -20849.624} C_VEL
LIN {X 0,Y 218.223,Z 335.749,A -85,B 0,C 180,E1 -20850.591,E2 -20850.591} C_VEL
LIN {X 0,Y 217.34,Z 334.167,A -85,B 0,C 180,E1 -20850.985,E2 -20850.985} C_VEL
LIN {X 0,Y 215.045,Z 332.111,A -85,B 0,C 180,E1 -20851.926,E2 -20851.926} C_VEL
LIN {X 0,Y 213.96,Z 329.781,A -85,B 0,C 180,E1 -20852.463,E2 -20852.463} C_VEL
LIN {X 0,Y 213.784,Z 328.855,A -85,B 0,C 180,E1 -20852.598,E2 -20852.598} C_VEL
LIN {X 0,Y 213.792,Z 328.846,A -85,B 0,C 180,E1 -20856.986,E2 -20856.986} C_VEL
LIN {X 0,Y 213.871,Z 328.832,A -85,B 0,C 180,E1 -20862.798,E2 -20862.798} C_VEL
LIN {X 0,Y 213.897,Z 328.824,A -85,B 0,C 180,E1 -20866.703,E2 -20866.703} C_VEL
LIN {X 0,Y 214.119,Z 328.798,A -85,B 0,C 180,E1 -20870.555,E2 -20870.555} C_VEL
LIN {X 0,Y 214.059,Z 328.819,A -85,B 0,C 180,E1 -20874.348,E2 -20874.348} C_VEL
LIN {X 0,Y 214.367,Z 328.77,A -85,B 0,C 180,E1 -20878.122,E2 -20878.122} C_VEL
LIN {X 0,Y 214.5,Z 328.764,A -85,B 0,C 180,E1 -20880,E2 -20880} C_VEL
LIN {X 0,Y 214.395,Z 328.76,A -85,B 0,C 180,E1 -20881.879,E2 -20881.879} C_VEL
LIN {X 0,Y 214.174,Z 328.785,A -85,B 0,C 180,E1 -20887.543,E2 -20887.543} C_VEL
LIN {X 0,Y 213.987,Z 328.822,A -85,B 0,C 180,E1 -20891.366,E2 -20891.366} C_VEL
LIN {X 0,Y 213.902,Z 328.833,A -85,B 0,C 180,E1 -20895.24,E2 -20895.24} C_VEL
LIN {X 0,Y 213.813,Z 328.834,A -85,B 0,C 180,E1 -20899.19,E2 -20899.19} C_VEL
LIN {X 0,Y 213.79,Z 328.837,A -85,B 0,C 180,E1 -20903.234,E2 -20903.234} C_VEL
LIN {X 0,Y 213.779,Z 328.842,A -85,B 0,C 180,E1 -20907.428,E2 -20907.428} C_VEL
LIN {X 0,Y 213.753,Z 328.848,A -85,B 0,C 180,E1 -20911.741,E2 -20911.741} C_VEL
LIN {X 0,Y 213.735,Z 328.854,A -85,B 0,C 180,E1 -20916.291,E2 -20916.291} C_VEL
LIN {X 0,Y 213.761,Z 328.941,A -85,B 0,C 180,E1 -20917.288,E2 -20917.288} C_VEL
LIN {X 0,Y 215.388,Z 334.196,A -85,B 0,C 180,E1 -20921.251,E2 -20921.251} C_VEL
LIN {X 0,Y 216.081,Z 336.027,A -85,B 0,C 180,E1 -20922.126,E2 -20922.126} C_VEL
LIN {X 0,Y 217.456,Z 339.285,A -85,B 0,C 180,E1 -20923,E2 -20923} C_VEL
LIN {X 0,Y 219.417,Z 344.824,A -85,B 0,C 180,E1 -20923.963,E2 -20923.963} C_VEL
LIN {X 0,Y 222.468,Z 355.392,A -85,B 0,C 180,E1 -20925.47,E2 -20925.47} C_VEL
LIN {X 0,Y 223.755,Z 358.655,A -85,B 0,C 180,E1 -20926.031,E2 -20926.031} C_VEL
LIN {X 0,Y 229.28,Z 368.473,A -85,B 0,C 180,E1 -20928.08,E2 -20928.08} C_VEL
LIN {X 0,Y 235.426,Z 380.908,A -85,B 0,C 180,E1 -20930.22,E2 -20930.22} C_VEL
LIN {X 0,Y 240.32,Z 392.226,A -85,B 0,C 180,E1 -20931.848,E2 -20931.848} C_VEL
LIN {X 0,Y 241.121,Z 397.94,A -85,B 0,C 180,E1 -20932.262,E2 -20932.262} C_VEL
LIN {X 0,Y 238.376,Z 446.011,A -85,B 0,C 180,E1 -20933.675,E2 -20933.675} C_VEL
LIN {X 0,Y 236.693,Z 459.505,A -85,B 0,C 180,E1 -20934.361,E2 -20934.361} C_VEL
LIN {X 0,Y 234.333,Z 471.784,A -85,B 0,C 180,E1 -20935.263,E2 -20935.263} C_VEL
LIN {X 0,Y 231.267,Z 484.343,A -85,B 0,C 180,E1 -20936.58,E2 -20936.58} C_VEL
LIN {X 0,Y 227.969,Z 495.54,A -85,B 0,C 180,E1 -20938.136,E2 -20938.136} C_VEL
LIN {X 0,Y 224.869,Z 504.619,A -85,B 0,C 180,E1 -20939.739,E2 -20939.739} C_VEL
LIN {X 0,Y 221.578,Z 513.113,A -85,B 0,C 180,E1 -20941.593,E2 -20941.593} C_VEL
LIN {X 0,Y 218.246,Z 520.966,A -85,B 0,C 180,E1 -20943.721,E2 -20943.721} C_VEL
LIN {X 0,Y 215.172,Z 527.737,A -85,B 0,C 180,E1 -20946.008,E2 -20946.008} C_VEL
LIN {X 0,Y 212.334,Z 533.944,A -85,B 0,C 180,E1 -20948.651,E2 -20948.651} C_VEL
LIN {X 0,Y 209.767,Z 539.1,A -85,B 0,C 180,E1 -20951.443,E2 -20951.443} C_VEL
LIN {X 0,Y 207.613,Z 543.125,A -85,B 0,C 180,E1 -20954.289,E2 -20954.289} C_VEL
LIN {X 0,Y 206.593,Z 545.224,A -85,B 0,C 180,E1 -20956.226,E2 -20956.226} C_VEL
LIN {X 0,Y 205.12,Z 548.185,A -85,B 0,C 180,E1 -20960.138,E2 -20960.138} C_VEL
LIN {X 0,Y 204.672,Z 549.083,A -85,B 0,C 180,E1 -20962.107,E2 -20962.107} C_VEL
LIN {X 0,Y 204.317,Z 549.641,A -85,B 0,C 180,E1 -20966.057,E2 -20966.057} C_VEL
LIN {X 0,Y 204.371,Z 549.344,A -85,B 0,C 180,E1 -20968.031,E2 -20968.031} C_VEL
LIN {X 0,Y 204.499,Z 548.663,A -85,B 0,C 180,E1 -20970.002,E2 -20970.002} C_VEL
LIN {X 0,Y 204.402,Z 547.544,A -85,B 0,C 180,E1 -20971.972,E2 -20971.972} C_VEL
LIN {X 0,Y 204.38,Z 545.691,A -85,B 0,C 180,E1 -20974.267,E2 -20974.267} C_VEL
LIN {X 0,Y 204.564,Z 542.832,A -85,B 0,C 180,E1 -20976.908,E2 -20976.908} C_VEL
LIN {X 0,Y 204.975,Z 538.589,A -85,B 0,C 180,E1 -20979.873,E2 -20979.873} C_VEL
LIN {X 0,Y 205.919,Z 532.113,A -85,B 0,C 180,E1 -20983.321,E2 -20983.321} C_VEL
LIN {X 0,Y 207.358,Z 525.027,A -85,B 0,C 180,E1 -20986.239,E2 -20986.239} C_VEL
LIN {X 0,Y 208.913,Z 517.78,A -85,B 0,C 180,E1 -20988.64,E2 -20988.64} C_VEL
LIN {X 0,Y 210.716,Z 508.014,A -85,B 0,C 180,E1 -20991.253,E2 -20991.253} C_VEL
LIN {X 0,Y 212.71,Z 498.08,A -85,B 0,C 180,E1 -20993.36,E2 -20993.36} C_VEL
LIN {X 0,Y 214.694,Z 487.212,A -85,B 0,C 180,E1 -20995.187,E2 -20995.187} C_VEL
LIN {X 0,Y 216.662,Z 474.992,A -85,B 0,C 180,E1 -20996.75,E2 -20996.75} C_VEL
LIN {X 0,Y 218.296,Z 462.2,A -85,B 0,C 180,E1 -20997.96,E2 -20997.96} C_VEL
LIN {X 0,Y 219.459,Z 449.786,A -85,B 0,C 180,E1 -20998.761,E2 -20998.761} C_VEL
LIN {X 0,Y 220.305,Z 432.926,A -85,B 0,C 180,E1 -20999.389,E2 -20999.389} C_VEL
LIN {X 0,Y 221.756,Z 390.074,A -85,B 0,C 180,E1 -21000.737,E2 -21000.737} C_VEL
LIN {X 0,Y 218.551,Z 363.364,A -85,B 0,C 180,E1 -21002.102,E2 -21002.102} C_VEL
LIN {X 0,Y 212.43,Z 346.882,A -85,B 0,C 180,E1 -21003.551,E2 -21003.551} C_VEL
LIN {X 0,Y 208.391,Z 337.139,A -85,B 0,C 180,E1 -21004.519,E2 -21004.519} C_VEL
LIN {X 0,Y 206.665,Z 329.744,A -85,B 0,C 180,E1 -21008.144,E2 -21008.144} C_VEL
LIN {X 0,Y 206.623,Z 329.75,A -85,B 0,C 180,E1 -21012.867,E2 -21012.867} C_VEL
LIN {X 0,Y 206.627,Z 329.75,A -85,B 0,C 180,E1 -21017.135,E2 -21017.135} C_VEL
LIN {X 0,Y 206.693,Z 329.735,A -85,B 0,C 180,E1 -21021.451,E2 -21021.451} C_VEL
LIN {X 0,Y 206.705,Z 329.736,A -85,B 0,C 180,E1 -21024.689,E2 -21024.689} C_VEL
LIN {X 0,Y 206.701,Z 329.736,A -85,B 0,C 180,E1 -21029.335,E2 -21029.335} C_VEL
LIN {X 0,Y 206.712,Z 329.734,A -85,B 0,C 180,E1 -21033.769,E2 -21033.769} C_VEL
LIN {X 0,Y 206.739,Z 329.723,A -85,B 0,C 180,E1 -21038.041,E2 -21038.041} C_VEL
LIN {X 0,Y 206.831,Z 329.714,A -85,B 0,C 180,E1 -21042.192,E2 -21042.192} C_VEL
LIN {X 0,Y 206.885,Z 329.711,A -85,B 0,C 180,E1 -21046.243,E2 -21046.243} C_VEL
LIN {X 0,Y 207.086,Z 329.663,A -85,B 0,C 180,E1 -21050.23,E2 -21050.23} C_VEL
LIN {X 0,Y 207.053,Z 329.687,A -85,B 0,C 180,E1 -21054.155,E2 -21054.155} C_VEL
LIN {X 0,Y 207.355,Z 329.651,A -85,B 0,C 180,E1 -21058.057,E2 -21058.057} C_VEL
LIN {X 0,Y 207.51,Z 329.622,A -85,B 0,C 180,E1 -21060,E2 -21060} C_VEL
LIN {X 0,Y 207.058,Z 329.669,A -85,B 0,C 180,E1 -21063.892,E2 -21063.892} C_VEL
LIN {X 0,Y 207.134,Z 329.68,A -85,B 0,C 180,E1 -21067.8,E2 -21067.8} C_VEL
LIN {X 0,Y 206.925,Z 329.702,A -85,B 0,C 180,E1 -21071.758,E2 -21071.758} C_VEL
LIN {X 0,Y 206.833,Z 329.692,A -85,B 0,C 180,E1 -21075.773,E2 -21075.773} C_VEL
LIN {X 0,Y 206.735,Z 329.729,A -85,B 0,C 180,E1 -21079.874,E2 -21079.874} C_VEL
LIN {X 0,Y 206.742,Z 329.725,A -85,B 0,C 180,E1 -21084.074,E2 -21084.074} C_VEL
LIN {X 0,Y 206.692,Z 329.712,A -85,B 0,C 180,E1 -21088.426,E2 -21088.426} C_VEL
LIN {X 0,Y 206.699,Z 329.733,A -85,B 0,C 180,E1 -21092.957,E2 -21092.957} C_VEL
LIN {X 0,Y 206.682,Z 329.715,A -85,B 0,C 180,E1 -21097.739,E2 -21097.739} C_VEL
LIN {X 0,Y 206.645,Z 329.737,A -85,B 0,C 180,E1 -21101.561,E2 -21101.561} C_VEL
LIN {X 0,Y 206.634,Z 329.737,A -85,B 0,C 180,E1 -21105.581,E2 -21105.581} C_VEL
LIN {X 0,Y 206.663,Z 329.735,A -85,B 0,C 180,E1 -21109.747,E2 -21109.747} C_VEL
LIN {X 0,Y 206.702,Z 329.724,A -85,B 0,C 180,E1 -21114.687,E2 -21114.687} C_VEL
LIN {X 0,Y 206.697,Z 329.735,A -85,B 0,C 180,E1 -21119.333,E2 -21119.333} C_VEL
LIN {X 0,Y 206.709,Z 329.736,A -85,B 0,C 180,E1 -21123.767,E2 -21123.767} C_VEL
LIN {X 0,Y 206.739,Z 329.734,A -85,B 0,C 180,E1 -21128.039,E2 -21128.039} C_VEL
LIN {X 0,Y 206.771,Z 329.731,A -85,B 0,C 180,E1 -21129.38,E2 -21129.38} C_VEL
LIN {X 0,Y 207.964,Z 332.817,A -85,B 0,C 180,E1 -21129.708,E2 -21129.708} C_VEL
LIN {X 0,Y 214.3,Z 345.225,A -85,B 0,C 180,E1 -21131.113,E2 -21131.113} C_VEL
LIN {X 0,Y 220.561,Z 361.96,A -85,B 0,C 180,E1 -21132.57,E2 -21132.57} C_VEL
LIN {X 0,Y 222.616,Z 368.399,A -85,B 0,C 180,E1 -21133.06,E2 -21133.06} C_VEL
LIN {X 0,Y 219.898,Z 434.567,A -85,B 0,C 180,E1 -21135.134,E2 -21135.134} C_VEL
LIN {X 0,Y 218.832,Z 447.647,A -85,B 0,C 180,E1 -21135.883,E2 -21135.883} C_VEL
LIN {X 0,Y 217.596,Z 459.753,A -85,B 0,C 180,E1 -21136.931,E2 -21136.931} C_VEL
LIN {X 0,Y 216.098,Z 471.194,A -85,B 0,C 180,E1 -21138.27,E2 -21138.27} C_VEL
LIN {X 0,Y 214.295,Z 482.035,A -85,B 0,C 180,E1 -21139.913,E2 -21139.913} C_VEL
LIN {X 0,Y 212.314,Z 492.449,A -85,B 0,C 180,E1 -21141.911,E2 -21141.911} C_VEL
LIN {X 0,Y 210.345,Z 502.15,A -85,B 0,C 180,E1 -21144.246,E2 -21144.246} C_VEL
LIN {X 0,Y 208.652,Z 510.101,A -85,B 0,C 180,E1 -21146.619,E2 -21146.619} C_VEL
LIN {X 0,Y 207.009,Z 517.866,A -85,B 0,C 180,E1 -21149.512,E2 -21149.512} C_VEL
LIN {X 0,Y 206.009,Z 523.167,A -85,B 0,C 180,E1 -21151.953,E2 -21151.953} C_VEL
LIN {X 0,Y 205.2,Z 528.299,A -85,B 0,C 180,E1 -21154.91,E2 -21154.91} C_VEL
LIN {X 0,Y 204.588,Z 532.296,A -85,B 0,C 180,E1 -21157.896,E2 -21157.896} C_VEL
LIN {X 0,Y 204.247,Z 534.362,A -85,B 0,C 180,E1 -21159.905,E2 -21159.905} C_VEL
LIN {X 0,Y 204.084,Z 536.004,A -85,B 0,C 180,E1 -21161.922,E2 -21161.922} C_VEL
LIN {X 0,Y 204.165,Z 537.842,A -85,B 0,C 180,E1 -21165.455,E2 -21165.455} C_VEL
LIN {X 0,Y 204.361,Z 538.347,A -85,B 0,C 180,E1 -21168.028,E2 -21168.028} C_VEL
LIN {X 0,Y 204.723,Z 538.309,A -85,B 0,C 180,E1 -21170.076,E2 -21170.076} C_VEL
LIN {X 0,Y 205.386,Z 537.677,A -85,B 0,C 180,E1 -21172.498,E2 -21172.498} C_VEL
LIN {X 0,Y 206.816,Z 535.56,A -85,B 0,C 180,E1 -21176.214,E2 -21176.214} C_VEL
LIN {X 0,Y 208.206,Z 533.321,A -85,B 0,C 180,E1 -21178.643,E2 -21178.643} C_VEL
LIN {X 0,Y 210.817,Z 528.661,A -85,B 0,C 180,E1 -21182.233,E2 -21182.233} C_VEL
LIN {X 0,Y 213.593,Z 523.415,A -85,B 0,C 180,E1 -21185.153,E2 -21185.153} C_VEL
LIN {X 0,Y 216.815,Z 516.69,A -85,B 0,C 180,E1 -21188.013,E2 -21188.013} C_VEL
LIN {X 0,Y 220.587,Z 508.248,A -85,B 0,C 180,E1 -21190.776,E2 -21190.776} C_VEL
LIN {X 0,Y 224.128,Z 499.546,A -85,B 0,C 180,E1 -21192.999,E2 -21192.999} C_VEL
LIN {X 0,Y 227.598,Z 489.851,A -85,B 0,C 180,E1 -21194.946,E2 -21194.946} C_VEL
LIN {X 0,Y 230.812,Z 479.262,A -85,B 0,C 180,E1 -21196.63,E2 -21196.63} C_VEL
LIN {X 0,Y 233.817,Z 467.56,A -85,B 0,C 180,E1 -21198.064,E2 -21198.064} C_VEL
LIN {X 0,Y 236.055,Z 456.602,A -85,B 0,C 180,E1 -21199.081,E2 -21199.081} C_VEL
LIN {X 0,Y 237.91,Z 443.59,A -85,B 0,C 180,E1 -21199.962,E2 -21199.962} C_VEL
LIN {X 0,Y 239.133,Z 430.599,A -85,B 0,C 180,E1 -21200.509,E2 -21200.509} C_VEL
LIN {X 0,Y 241.655,Z 386.927,A -85,B 0,C 180,E1 -21201.73,E2 -21201.73} C_VEL
LIN {X 0,Y 236.1,Z 375.019,A -85,B 0,C 180,E1 -21203.531,E2 -21203.531} C_VEL
LIN {X 0,Y 228.916,Z 361.691,A -85,B 0,C 180,E1 -21205.998,E2 -21205.998} C_VEL
LIN {X 0,Y 222.763,Z 351.815,A -85,B 0,C 180,E1 -21208.274,E2 -21208.274} C_VEL
LIN {X 0,Y 220.263,Z 348.356,A -85,B 0,C 180,E1 -21209.24,E2 -21209.24} C_VEL
LIN {X 0,Y 217.448,Z 344.512,A -85,B 0,C 180,E1 -21210.386,E2 -21210.386} C_VEL
LIN {X 0,Y 214.761,Z 340.806,A -85,B 0,C 180,E1 -21211.54,E2 -21211.54} C_VEL
LIN {X 0,Y 211.556,Z 337.068,A -85,B 0,C 180,E1 -21212.959,E2 -21212.959} C_VEL
LIN {X 0,Y 210.484,Z 335.15,A -85,B 0,C 180,E1 -21213.496,E2 -21213.496} C_VEL
LIN {X 0,Y 208.154,Z 333.197,A -85,B 0,C 180,E1 -21214.569,E2 -21214.569} C_VEL
LIN {X 0,Y 206.881,Z 330.627,A -85,B 0,C 180,E1 -21215.275,E2 -21215.275} C_VEL
LIN {X 0,Y 206.703,Z 329.734,A -85,B 0,C 180,E1 -21215.453,E2 -21215.453} C_VEL
LIN {X 0,Y 206.705,Z 329.737,A -85,B 0,C 180,E1 -21220.124,E2 -21220.124} C_VEL
LIN {X 0,Y 206.797,Z 329.726,A -85,B 0,C 180,E1 -21224.224,E2 -21224.224} C_VEL
LIN {X 0,Y 207.054,Z 329.685,A -85,B 0,C 180,E1 -21229.835,E2 -21229.835} C_VEL
LIN {X 0,Y 207.113,Z 329.668,A -85,B 0,C 180,E1 -21232.199,E2 -21232.199} C_VEL
LIN {X 0,Y 207.309,Z 329.648,A -85,B 0,C 180,E1 -21238.058,E2 -21238.058} C_VEL
LIN {X 0,Y 207.468,Z 329.64,A -85,B 0,C 180,E1 -21240,E2 -21240} C_VEL
LIN {X 0,Y 207.334,Z 329.639,A -85,B 0,C 180,E1 -21241.943,E2 -21241.943} C_VEL
LIN {X 0,Y 207.118,Z 329.663,A -85,B 0,C 180,E1 -21247.801,E2 -21247.801} C_VEL
LIN {X 0,Y 206.909,Z 329.697,A -85,B 0,C 180,E1 -21251.76,E2 -21251.76} C_VEL
LIN {X 0,Y 206.837,Z 329.716,A -85,B 0,C 180,E1 -21255.774,E2 -21255.774} C_VEL
LIN {X 0,Y 206.85,Z 329.698,A -85,B 0,C 180,E1 -21257.956,E2 -21257.956} C_VEL
LIN {X 0,Y 206.732,Z 329.716,A -85,B 0,C 180,E1 -21263.387,E2 -21263.387} C_VEL
LIN {X 0,Y 206.681,Z 329.728,A -85,B 0,C 180,E1 -21268.429,E2 -21268.429} C_VEL
LIN {X 0,Y 206.688,Z 329.733,A -85,B 0,C 180,E1 -21272.96,E2 -21272.96} C_VEL
LIN {X 0,Y 206.733,Z 329.887,A -85,B 0,C 180,E1 -21274.924,E2 -21274.924} C_VEL
LIN {X 0,Y 208.495,Z 335.352,A -85,B 0,C 180,E1 -21279.371,E2 -21279.371} C_VEL
LIN {X 0,Y 211.51,Z 339.964,A -85,B 0,C 180,E1 -21280.858,E2 -21280.858} C_VEL
LIN {X 0,Y 213.138,Z 342.072,A -85,B 0,C 180,E1 -21281.599,E2 -21281.599} C_VEL
LIN {X 0,Y 217.352,Z 348.443,A -85,B 0,C 180,E1 -21283.459,E2 -21283.459} C_VEL
LIN {X 0,Y 220.996,Z 354.228,A -85,B 0,C 180,E1 -21284.959,E2 -21284.959} C_VEL
LIN {X 0,Y 223.755,Z 358.655,A -85,B 0,C 180,E1 -21286.031,E2 -21286.031} C_VEL
LIN {X 0,Y 226.087,Z 365.099,A -85,B 0,C 180,E1 -21287.028,E2 -21287.028} C_VEL
LIN {X 0,Y 229.464,Z 379.286,A -85,B 0,C 180,E1 -21288.625,E2 -21288.625} C_VEL
LIN {X 0,Y 231.555,Z 386.147,A -85,B 0,C 180,E1 -21289.48,E2 -21289.48} C_VEL
LIN {X 0,Y 235.433,Z 395.387,A -85,B 0,C 180,E1 -21290.841,E2 -21290.841} C_VEL
LIN {X 0,Y 235.911,Z 399.723,A -85,B 0,C 180,E1 -21291.139,E2 -21291.139} C_VEL
LIN {X 0,Y 233.18,Z 445.256,A -85,B 0,C 180,E1 -21292.481,E2 -21292.481} C_VEL
LIN {X 0,Y 231.531,Z 458.657,A -85,B 0,C 180,E1 -21293.168,E2 -21293.168} C_VEL
LIN {X 0,Y 229.074,Z 471.127,A -85,B 0,C 180,E1 -21294.075,E2 -21294.075} C_VEL
LIN {X 0,Y 226.321,Z 482.243,A -85,B 0,C 180,E1 -21295.21,E2 -21295.21} C_VEL
LIN {X 0,Y 222.88,Z 493.78,A -85,B 0,C 180,E1 -21296.781,E2 -21296.781} C_VEL
LIN {X 0,Y 219.591,Z 503.125,A -85,B 0,C 180,E1 -21298.396,E2 -21298.396} C_VEL
LIN {X 0,Y 215.384,Z 513.593,A -85,B 0,C 180,E1 -21300.698,E2 -21300.698} C_VEL
LIN {X 0,Y 211.252,Z 522.672,A -85,B 0,C 180,E1 -21303.315,E2 -21303.315} C_VEL
LIN {X 0,Y 207.751,Z 530.005,A -85,B 0,C 180,E1 -21306.052,E2 -21306.052} C_VEL
LIN {X 0,Y 204.792,Z 535.915,A -85,B 0,C 180,E1 -21308.881,E2 -21308.881} C_VEL
LIN {X 0,Y 202.227,Z 540.608,A -85,B 0,C 180,E1 -21311.775,E2 -21311.775} C_VEL
LIN {X 0,Y 200.192,Z 544.215,A -85,B 0,C 180,E1 -21314.736,E2 -21314.736} C_VEL
LIN {X 0,Y 198.777,Z 546.839,A -85,B 0,C 180,E1 -21317.754,E2 -21317.754} C_VEL
LIN {X 0,Y 197.641,Z 548.942,A -85,B 0,C 180,E1 -21321.825,E2 -21321.825} C_VEL
LIN {X 0,Y 197.247,Z 549.426,A -85,B 0,C 180,E1 -21325.915,E2 -21325.915} C_VEL
LIN {X 0,Y 197.274,Z 549.099,A -85,B 0,C 180,E1 -21327.96,E2 -21327.96} C_VEL
LIN {X 0,Y 197.417,Z 548.383,A -85,B 0,C 180,E1 -21330.002,E2 -21330.002} C_VEL
LIN {X 0,Y 197.306,Z 547.207,A -85,B 0,C 180,E1 -21332.043,E2 -21332.043} C_VEL
LIN {X 0,Y 197.33,Z 544.672,A -85,B 0,C 180,E1 -21335.11,E2 -21335.11} C_VEL
LIN {X 0,Y 197.594,Z 541.101,A -85,B 0,C 180,E1 -21338.181,E2 -21338.181} C_VEL
LIN {X 0,Y 198.181,Z 536.393,A -85,B 0,C 180,E1 -21341.249,E2 -21341.249} C_VEL
LIN {X 0,Y 199.431,Z 529.276,A -85,B 0,C 180,E1 -21344.805,E2 -21344.805} C_VEL
LIN {X 0,Y 201.039,Z 521.542,A -85,B 0,C 180,E1 -21347.813,E2 -21347.813} C_VEL
LIN {X 0,Y 202.758,Z 513.598,A -85,B 0,C 180,E1 -21350.282,E2 -21350.282} C_VEL
LIN {X 0,Y 204.725,Z 503.865,A -85,B 0,C 180,E1 -21352.72,E2 -21352.72} C_VEL
LIN {X 0,Y 206.902,Z 493.065,A -85,B 0,C 180,E1 -21354.858,E2 -21354.858} C_VEL
LIN {X 0,Y 208.868,Z 482.61,A -85,B 0,C 180,E1 -21356.479,E2 -21356.479} C_VEL
LIN {X 0,Y 210.77,Z 470.01,A -85,B 0,C 180,E1 -21357.965,E2 -21357.965} C_VEL
LIN {X 0,Y 212.278,Z 456.678,A -85,B 0,C 180,E1 -21359.097,E2 -21359.097} C_VEL
LIN {X 0,Y 213.269,Z 444.645,A -85,B 0,C 180,E1 -21359.759,E2 -21359.759} C_VEL
LIN {X 0,Y 215.292,Z 390.628,A -85,B 0,C 180,E1 -21361.526,E2 -21361.526} C_VEL
LIN {X 0,Y 212.485,Z 365.881,A -85,B 0,C 180,E1 -21362.825,E2 -21362.825} C_VEL
LIN {X 0,Y 206.745,Z 350.276,A -85,B 0,C 180,E1 -21364.255,E2 -21364.255} C_VEL
LIN {X 0,Y 201.098,Z 336.828,A -85,B 0,C 180,E1 -21365.717,E2 -21365.717} C_VEL
LIN {X 0,Y 199.617,Z 330.622,A -85,B 0,C 180,E1 -21368.951,E2 -21368.951} C_VEL
LIN {X 0,Y 199.571,Z 330.632,A -85,B 0,C 180,E1 -21372.308,E2 -21372.308} C_VEL
LIN {X 0,Y 199.582,Z 330.628,A -85,B 0,C 180,E1 -21375.228,E2 -21375.228} C_VEL
LIN {X 0,Y 199.583,Z 330.627,A -85,B 0,C 180,E1 -21378.005,E2 -21378.005} C_VEL
LIN {X 0,Y 199.615,Z 330.62,A -85,B 0,C 180,E1 -21380.768,E2 -21380.768} C_VEL
LIN {X 0,Y 199.616,Z 330.618,A -85,B 0,C 180,E1 -21385.714,E2 -21385.714} C_VEL
LIN {X 0,Y 199.691,Z 330.609,A -85,B 0,C 180,E1 -21388.135,E2 -21388.135} C_VEL
LIN {X 0,Y 199.65,Z 330.613,A -85,B 0,C 180,E1 -21392.766,E2 -21392.766} C_VEL
LIN {X 0,Y 199.713,Z 330.602,A -85,B 0,C 180,E1 -21397.226,E2 -21397.226} C_VEL
LIN {X 0,Y 199.755,Z 330.59,A -85,B 0,C 180,E1 -21401.799,E2 -21401.799} C_VEL
LIN {X 0,Y 199.822,Z 330.593,A -85,B 0,C 180,E1 -21405.747,E2 -21405.747} C_VEL
LIN {X 0,Y 200.029,Z 330.542,A -85,B 0,C 180,E1 -21409.882,E2 -21409.882} C_VEL
LIN {X 0,Y 200.016,Z 330.561,A -85,B 0,C 180,E1 -21413.949,E2 -21413.949} C_VEL
LIN {X 0,Y 200.297,Z 330.531,A -85,B 0,C 180,E1 -21417.989,E2 -21417.989} C_VEL
LIN {X 0,Y 200.475,Z 330.497,A -85,B 0,C 180,E1 -21420,E2 -21420} C_VEL
LIN {X 0,Y 200.003,Z 330.547,A -85,B 0,C 180,E1 -21424.03,E2 -21424.03} C_VEL
LIN {X 0,Y 200.082,Z 330.56,A -85,B 0,C 180,E1 -21428.076,E2 -21428.076} C_VEL
LIN {X 0,Y 199.873,Z 330.576,A -85,B 0,C 180,E1 -21432.179,E2 -21432.179} C_VEL
LIN {X 0,Y 199.769,Z 330.573,A -85,B 0,C 180,E1 -21436.346,E2 -21436.346} C_VEL
LIN {X 0,Y 199.666,Z 330.611,A -85,B 0,C 180,E1 -21440.608,E2 -21440.608} C_VEL
LIN {X 0,Y 199.655,Z 330.6,A -85,B 0,C 180,E1 -21444.986,E2 -21444.986} C_VEL
LIN {X 0,Y 199.612,Z 330.599,A -85,B 0,C 180,E1 -21449.532,E2 -21449.532} C_VEL
LIN {X 0,Y 199.669,Z 330.608,A -85,B 0,C 180,E1 -21452.351,E2 -21452.351} C_VEL
LIN {X 0,Y 199.626,Z 330.601,A -85,B 0,C 180,E1 -21456.762,E2 -21456.762} C_VEL
LIN {X 0,Y 199.61,Z 330.596,A -85,B 0,C 180,E1 -21459.327,E2 -21459.327} C_VEL
LIN {X 0,Y 199.577,Z 330.622,A -85,B 0,C 180,E1 -21462.309,E2 -21462.309} C_VEL
LIN {X 0,Y 199.581,Z 330.619,A -85,B 0,C 180,E1 -21465.227,E2 -21465.227} C_VEL
LIN {X 0,Y 199.58,Z 330.606,A -85,B 0,C 180,E1 -21468.003,E2 -21468.003} C_VEL
LIN {X 0,Y 199.613,Z 330.619,A -85,B 0,C 180,E1 -21470.766,E2 -21470.766} C_VEL
LIN {X 0,Y 199.612,Z 330.608,A -85,B 0,C 180,E1 -21475.712,E2 -21475.712} C_VEL
LIN {X 0,Y 199.688,Z 330.612,A -85,B 0,C 180,E1 -21478.133,E2 -21478.133} C_VEL
LIN {X 0,Y 199.647,Z 330.617,A -85,B 0,C 180,E1 -21482.764,E2 -21482.764} C_VEL
LIN {X 0,Y 199.71,Z 330.61,A -85,B 0,C 180,E1 -21487.844,E2 -21487.844} C_VEL
LIN {X 0,Y 199.725,Z 330.747,A -85,B 0,C 180,E1 -21488.305,E2 -21488.305} C_VEL
LIN {X 0,Y 200.805,Z 333.589,A -85,B 0,C 180,E1 -21488.602,E2 -21488.602} C_VEL
LIN {X 0,Y 208.17,Z 347.54,A -85,B 0,C 180,E1 -21490.313,E2 -21490.313} C_VEL
LIN {X 0,Y 214.116,Z 363.291,A -85,B 0,C 180,E1 -21491.764,E2 -21491.764} C_VEL
LIN {X 0,Y 216.179,Z 370.01,A -85,B 0,C 180,E1 -21492.292,E2 -21492.292} C_VEL
LIN {X 0,Y 213.414,Z 434.978,A -85,B 0,C 180,E1 -21494.387,E2 -21494.387} C_VEL
LIN {X 0,Y 212.325,Z 447.734,A -85,B 0,C 180,E1 -21495.134,E2 -21495.134} C_VEL
LIN {X 0,Y 210.965,Z 460.433,A -85,B 0,C 180,E1 -21496.268,E2 -21496.268} C_VEL
LIN {X 0,Y 209.414,Z 471.745,A -85,B 0,C 180,E1 -21497.645,E2 -21497.645} C_VEL
LIN {X 0,Y 207.551,Z 482.428,A -85,B 0,C 180,E1 -21499.319,E2 -21499.319} C_VEL
LIN {X 0,Y 205.488,Z 492.875,A -85,B 0,C 180,E1 -21501.393,E2 -21501.393} C_VEL
LIN {X 0,Y 203.658,Z 501.638,A -85,B 0,C 180,E1 -21503.559,E2 -21503.559} C_VEL
LIN {X 0,Y 201.852,Z 509.71,A -85,B 0,C 180,E1 -21506.005,E2 -21506.005} C_VEL
LIN {X 0,Y 200.103,Z 517.621,A -85,B 0,C 180,E1 -21508.992,E2 -21508.992} C_VEL
LIN {X 0,Y 198.841,Z 523.925,A -85,B 0,C 180,E1 -21512.024,E2 -21512.024} C_VEL
LIN {X 0,Y 198.062,Z 528.829,A -85,B 0,C 180,E1 -21515.012,E2 -21515.012} C_VEL
LIN {X 0,Y 197.432,Z 532.827,A -85,B 0,C 180,E1 -21518.184,E2 -21518.184} C_VEL
LIN {X 0,Y 197.114,Z 534.841,A -85,B 0,C 180,E1 -21520.267,E2 -21520.267} C_VEL
LIN {X 0,Y 196.989,Z 536.43,A -85,B 0,C 180,E1 -21522.359,E2 -21522.359} C_VEL
LIN {X 0,Y 197.092,Z 538.037,A -85,B 0,C 180,E1 -21525.684,E2 -21525.684} C_VEL
LIN {X 0,Y 197.356,Z 538.577,A -85,B 0,C 180,E1 -21528.691,E2 -21528.691} C_VEL
LIN {X 0,Y 197.792,Z 538.469,A -85,B 0,C 180,E1 -21530.811,E2 -21530.811} C_VEL
LIN {X 0,Y 198.405,Z 537.904,A -85,B 0,C 180,E1 -21532.93,E2 -21532.93} C_VEL
LIN {X 0,Y 199.175,Z 536.929,A -85,B 0,C 180,E1 -21535.049,E2 -21535.049} C_VEL
LIN {X 0,Y 200.166,Z 535.531,A -85,B 0,C 180,E1 -21537.155,E2 -21537.155} C_VEL
LIN {X 0,Y 202.031,Z 532.644,A -85,B 0,C 180,E1 -21540.174,E2 -21540.174} C_VEL
LIN {X 0,Y 204.536,Z 528.394,A -85,B 0,C 180,E1 -21543.349,E2 -21543.349} C_VEL
LIN {X 0,Y 208.099,Z 521.94,A -85,B 0,C 180,E1 -21546.829,E2 -21546.829} C_VEL
LIN {X 0,Y 211.845,Z 514.396,A -85,B 0,C 180,E1 -21549.892,E2 -21549.892} C_VEL
LIN {X 0,Y 215.742,Z 505.835,A -85,B 0,C 180,E1 -21552.525,E2 -21552.525} C_VEL
LIN {X 0,Y 219.544,Z 496.521,A -85,B 0,C 180,E1 -21554.767,E2 -21554.767} C_VEL
LIN {X 0,Y 223.241,Z 486.16,A -85,B 0,C 180,E1 -21556.717,E2 -21556.717} C_VEL
LIN {X 0,Y 226.669,Z 474.478,A -85,B 0,C 180,E1 -21558.415,E2 -21558.415} C_VEL
LIN {X 0,Y 229.623,Z 462.294,A -85,B 0,C 180,E1 -21559.749,E2 -21559.749} C_VEL
LIN {X 0,Y 231.907,Z 449.318,A -85,B 0,C 180,E1 -21560.783,E2 -21560.783} C_VEL
LIN {X 0,Y 233.506,Z 435.939,A -85,B 0,C 180,E1 -21561.491,E2 -21561.491} C_VEL
LIN {X 0,Y 236.43,Z 389.332,A -85,B 0,C 180,E1 -21562.841,E2 -21562.841} C_VEL
LIN {X 0,Y 230.53,Z 376.741,A -85,B 0,C 180,E1 -21564.871,E2 -21564.871} C_VEL
LIN {X 0,Y 223.555,Z 364.059,A -85,B 0,C 180,E1 -21567.428,E2 -21567.428} C_VEL
LIN {X 0,Y 218.392,Z 355.741,A -85,B 0,C 180,E1 -21569.468,E2 -21569.468} C_VEL
LIN {X 0,Y 214.142,Z 349.997,A -85,B 0,C 180,E1 -21571.249,E2 -21571.249} C_VEL
LIN {X 0,Y 211.039,Z 345.815,A -85,B 0,C 180,E1 -21572.645,E2 -21572.645} C_VEL
LIN {X 0,Y 208.321,Z 342.272,A -85,B 0,C 180,E1 -21573.938,E2 -21573.938} C_VEL
LIN {X 0,Y 207.384,Z 341.083,A -85,B 0,C 180,E1 -21574.401,E2 -21574.401} C_VEL
LIN {X 0,Y 204.935,Z 338.354,A -85,B 0,C 180,E1 -21575.632,E2 -21575.632} C_VEL
LIN {X 0,Y 203.873,Z 336.228,A -85,B 0,C 180,E1 -21576.252,E2 -21576.252} C_VEL
LIN {X 0,Y 201.274,Z 334.295,A -85,B 0,C 180,E1 -21577.616,E2 -21577.616} C_VEL
LIN {X 0,Y 199.921,Z 331.848,A -85,B 0,C 180,E1 -21578.475,E2 -21578.475} C_VEL
LIN {X 0,Y 199.656,Z 330.606,A -85,B 0,C 180,E1 -21578.783,E2 -21578.783} C_VEL
LIN {X 0,Y 199.738,Z 330.59,A -85,B 0,C 180,E1 -21581.803,E2 -21581.803} C_VEL
LIN {X 0,Y 199.76,Z 330.587,A -85,B 0,C 180,E1 -21585.743,E2 -21585.743} C_VEL
LIN {X 0,Y 200.015,Z 330.561,A -85,B 0,C 180,E1 -21589.882,E2 -21589.882} C_VEL
LIN {X 0,Y 199.988,Z 330.572,A -85,B 0,C 180,E1 -21593.949,E2 -21593.949} C_VEL
LIN {X 0,Y 200.254,Z 330.526,A -85,B 0,C 180,E1 -21597.989,E2 -21597.989} C_VEL
LIN {X 0,Y 200.434,Z 330.516,A -85,B 0,C 180,E1 -21600,E2 -21600} C_VEL
LIN {X 0,Y 199.976,Z 330.566,A -85,B 0,C 180,E1 -21604.031,E2 -21604.031} C_VEL
LIN {X 0,Y 200.067,Z 330.542,A -85,B 0,C 180,E1 -21608.078,E2 -21608.078} C_VEL
LIN {X 0,Y 199.859,Z 330.571,A -85,B 0,C 180,E1 -21612.181,E2 -21612.181} C_VEL
LIN {X 0,Y 199.781,Z 330.591,A -85,B 0,C 180,E1 -21616.346,E2 -21616.346} C_VEL
LIN {X 0,Y 199.666,Z 330.61,A -85,B 0,C 180,E1 -21620.609,E2 -21620.609} C_VEL
LIN {X 0,Y 199.637,Z 330.613,A -85,B 0,C 180,E1 -21624.99,E2 -21624.99} C_VEL
LIN {X 0,Y 199.603,Z 330.621,A -85,B 0,C 180,E1 -21629.535,E2 -21629.535} C_VEL
LIN {X 0,Y 199.691,Z 330.814,A -85,B 0,C 180,E1 -21632.159,E2 -21632.159} C_VEL
LIN {X 0,Y 201.077,Z 335.016,A -85,B 0,C 180,E1 -21636.003,E2 -21636.003} C_VEL
LIN {X 0,Y 204.443,Z 339.9,A -85,B 0,C 180,E1 -21637.914,E2 -21637.914} C_VEL
LIN {X 0,Y 206.01,Z 341.849,A -85,B 0,C 180,E1 -21638.729,E2 -21638.729} C_VEL
LIN {X 0,Y 210.426,Z 348.324,A -85,B 0,C 180,E1 -21640.93,E2 -21640.93} C_VEL
LIN {X 0,Y 214.085,Z 353.869,A -85,B 0,C 180,E1 -21642.611,E2 -21642.611} C_VEL
LIN {X 0,Y 217.705,Z 359.822,A -85,B 0,C 180,E1 -21644.184,E2 -21644.184} C_VEL
LIN {X 0,Y 222.443,Z 367.703,A -85,B 0,C 180,E1 -21646.082,E2 -21646.082} C_VEL
LIN {X 0,Y 228.664,Z 379.843,A -85,B 0,C 180,E1 -21648.436,E2 -21648.436} C_VEL
LIN {X 0,Y 231.555,Z 386.147,A -85,B 0,C 180,E1 -21649.48,E2 -21649.48} C_VEL
LIN {X 0,Y 232.44,Z 389.623,A -85,B 0,C 180,E1 -21649.858,E2 -21649.858} C_VEL
LIN {X 0,Y 232.71,Z 395.375,A -85,B 0,C 180,E1 -21650.176,E2 -21650.176} C_VEL
LIN {X 0,Y 232.131,Z 401.312,A -85,B 0,C 180,E1 -21650.292,E2 -21650.292} C_VEL
LIN {X 0,Y 230.143,Z 413.684,A -85,B 0,C 180,E1 -21650.339,E2 -21650.339} C_VEL
LIN {X 0,Y 229.773,Z 417.816,A -85,B 0,C 180,E1 -21650.428,E2 -21650.428} C_VEL
LIN {X 0,Y 227.926,Z 446.288,A -85,B 0,C 180,E1 -21651.315,E2 -21651.315} C_VEL
LIN {X 0,Y 226.185,Z 459.33,A -85,B 0,C 180,E1 -21652.006,E2 -21652.006} C_VEL
LIN {X 0,Y 223.66,Z 471.539,A -85,B 0,C 180,E1 -21652.923,E2 -21652.923} C_VEL
LIN {X 0,Y 220.589,Z 483.279,A -85,B 0,C 180,E1 -21654.169,E2 -21654.169} C_VEL
LIN {X 0,Y 217.022,Z 494.592,A -85,B 0,C 180,E1 -21655.762,E2 -21655.762} C_VEL
LIN {X 0,Y 213.992,Z 502.706,A -85,B 0,C 180,E1 -21657.189,E2 -21657.189} C_VEL
LIN {X 0,Y 210.016,Z 512.329,A -85,B 0,C 180,E1 -21659.317,E2 -21659.317} C_VEL
LIN {X 0,Y 206.356,Z 520.24,A -85,B 0,C 180,E1 -21661.525,E2 -21661.525} C_VEL
LIN {X 0,Y 202.419,Z 528.023,A -85,B 0,C 180,E1 -21664.282,E2 -21664.282} C_VEL
LIN {X 0,Y 199.171,Z 534.261,A -85,B 0,C 180,E1 -21667.163,E2 -21667.163} C_VEL
LIN {X 0,Y 196.349,Z 539.256,A -85,B 0,C 180,E1 -21670.123,E2 -21670.123} C_VEL
LIN {X 0,Y 193.959,Z 543.148,A -85,B 0,C 180,E1 -21673.152,E2 -21673.152} C_VEL
LIN {X 0,Y 191.813,Z 546.778,A -85,B 0,C 180,E1 -21677.302,E2 -21677.302} C_VEL
LIN {X 0,Y 191.088,Z 547.997,A -85,B 0,C 180,E1 -21679.405,E2 -21679.405} C_VEL
LIN {X 0,Y 190.287,Z 549.189,A -85,B 0,C 180,E1 -21683.64,E2 -21683.64} C_VEL
LIN {X 0,Y 190.162,Z 549.181,A -85,B 0,C 180,E1 -21686.265,E2 -21686.265} C_VEL
LIN {X 0,Y 190.336,Z 548.084,A -85,B 0,C 180,E1 -21690.002,E2 -21690.002} C_VEL
LIN {X 0,Y 190.18,Z 545.601,A -85,B 0,C 180,E1 -21693.818,E2 -21693.818} C_VEL
LIN {X 0,Y 190.43,Z 541.959,A -85,B 0,C 180,E1 -21697.424,E2 -21697.424} C_VEL
LIN {X 0,Y 190.941,Z 537.573,A -85,B 0,C 180,E1 -21700.607,E2 -21700.607} C_VEL
LIN {X 0,Y 191.831,Z 531.961,A -85,B 0,C 180,E1 -21703.778,E2 -21703.778} C_VEL
LIN {X 0,Y 193.385,Z 524.949,A -85,B 0,C 180,E1 -21706.904,E2 -21706.904} C_VEL
LIN {X 0,Y 195.05,Z 517.769,A -85,B 0,C 180,E1 -21709.471,E2 -21709.471} C_VEL
LIN {X 0,Y 196.829,Z 509.025,A -85,B 0,C 180,E1 -21712.02,E2 -21712.02} C_VEL
LIN {X 0,Y 199.148,Z 498.251,A -85,B 0,C 180,E1 -21714.5,E2 -21714.5} C_VEL
LIN {X 0,Y 201.281,Z 487.538,A -85,B 0,C 180,E1 -21716.437,E2 -21716.437} C_VEL
LIN {X 0,Y 203.375,Z 475.552,A -85,B 0,C 180,E1 -21718.09,E2 -21718.09} C_VEL
LIN {X 0,Y 205.133,Z 463.056,A -85,B 0,C 180,E1 -21719.366,E2 -21719.366} C_VEL
LIN {X 0,Y 206.466,Z 450.134,A -85,B 0,C 180,E1 -21720.281,E2 -21720.281} C_VEL
LIN {X 0,Y 207.293,Z 435.962,A -85,B 0,C 180,E1 -21720.868,E2 -21720.868} C_VEL
LIN {X 0,Y 208.894,Z 391.179,A -85,B 0,C 180,E1 -21722.361,E2 -21722.361} C_VEL
LIN {X 0,Y 206.246,Z 367.717,A -85,B 0,C 180,E1 -21723.647,E2 -21723.647} C_VEL
LIN {X 0,Y 200.42,Z 351.979,A -85,B 0,C 180,E1 -21725.171,E2 -21725.171} C_VEL
LIN {X 0,Y 193.787,Z 336.612,A -85,B 0,C 180,E1 -21726.972,E2 -21726.972} C_VEL
LIN {X 0,Y 192.54,Z 331.504,A -85,B 0,C 180,E1 -21729.737,E2 -21729.737} C_VEL
LIN {X 0,Y 192.492,Z 331.511,A -85,B 0,C 180,E1 -21733.926,E2 -21733.926} C_VEL
LIN {X 0,Y 192.518,Z 331.506,A -85,B 0,C 180,E1 -21738.92,E2 -21738.92} C_VEL
LIN {X 0,Y 192.592,Z 331.495,A -85,B 0,C 180,E1 -21743.403,E2 -21743.403} C_VEL
LIN {X 0,Y 192.611,Z 331.493,A -85,B 0,C 180,E1 -21747.061,E2 -21747.061} C_VEL
LIN {X 0,Y 192.627,Z 331.488,A -85,B 0,C 180,E1 -21751.685,E2 -21751.685} C_VEL
LIN {X 0,Y 192.685,Z 331.481,A -85,B 0,C 180,E1 -21756.345,E2 -21756.345} C_VEL
LIN {X 0,Y 192.703,Z 331.464,A -85,B 0,C 180,E1 -21761.489,E2 -21761.489} C_VEL
LIN {X 0,Y 192.747,Z 331.475,A -85,B 0,C 180,E1 -21765.212,E2 -21765.212} C_VEL
LIN {X 0,Y 192.951,Z 331.425,A -85,B 0,C 180,E1 -21769.567,E2 -21769.567} C_VEL
LIN {X 0,Y 192.979,Z 331.436,A -85,B 0,C 180,E1 -21773.727,E2 -21773.727} C_VEL
LIN {X 0,Y 193.241,Z 331.41,A -85,B 0,C 180,E1 -21777.915,E2 -21777.915} C_VEL
LIN {X 0,Y 193.439,Z 331.373,A -85,B 0,C 180,E1 -21780,E2 -21780} C_VEL
LIN {X 0,Y 192.95,Z 331.426,A -85,B 0,C 180,E1 -21784.177,E2 -21784.177} C_VEL
LIN {X 0,Y 193.032,Z 331.44,A -85,B 0,C 180,E1 -21788.373,E2 -21788.373} C_VEL
LIN {X 0,Y 192.799,Z 331.452,A -85,B 0,C 180,E1 -21792.633,E2 -21792.633} C_VEL
LIN {X 0,Y 192.722,Z 331.454,A -85,B 0,C 180,E1 -21796.961,E2 -21796.961} C_VEL
LIN {X 0,Y 192.605,Z 331.492,A -85,B 0,C 180,E1 -21801.4,E2 -21801.4} C_VEL
LIN {X 0,Y 192.644,Z 331.481,A -85,B 0,C 180,E1 -21804.207,E2 -21804.207} C_VEL
LIN {X 0,Y 192.605,Z 331.466,A -85,B 0,C 180,E1 -21808.864,E2 -21808.864} C_VEL
LIN {X 0,Y 192.598,Z 331.491,A -85,B 0,C 180,E1 -21813.185,E2 -21813.185} C_VEL
LIN {X 0,Y 192.554,Z 331.471,A -85,B 0,C 180,E1 -21818.351,E2 -21818.351} C_VEL
LIN {X 0,Y 192.494,Z 331.504,A -85,B 0,C 180,E1 -21823.094,E2 -21823.094} C_VEL
LIN {X 0,Y 192.492,Z 331.489,A -85,B 0,C 180,E1 -21826.903,E2 -21826.903} C_VEL
LIN {X 0,Y 192.554,Z 331.5,A -85,B 0,C 180,E1 -21831.647,E2 -21831.647} C_VEL
LIN {X 0,Y 192.597,Z 331.489,A -85,B 0,C 180,E1 -21836.812,E2 -21836.812} C_VEL
LIN {X 0,Y 192.623,Z 331.49,A -85,B 0,C 180,E1 -21841.683,E2 -21841.683} C_VEL
LIN {X 0,Y 192.67,Z 331.487,A -85,B 0,C 180,E1 -21847.083,E2 -21847.083} C_VEL
LIN {X 0,Y 193.687,Z 334.35,A -85,B 0,C 180,E1 -21847.412,E2 -21847.412} C_VEL
LIN {X 0,Y 199.574,Z 345.117,A -85,B 0,C 180,E1 -21848.874,E2 -21848.874} C_VEL
LIN {X 0,Y 203.712,Z 353.865,A -85,B 0,C 180,E1 -21849.888,E2 -21849.888} C_VEL
LIN {X 0,Y 209.662,Z 370.628,A -85,B 0,C 180,E1 -21851.422,E2 -21851.422} C_VEL
LIN {X 0,Y 207.881,Z 416.682,A -85,B 0,C 180,E1 -21852.938,E2 -21852.938} C_VEL
LIN {X 0,Y 206.784,Z 436.985,A -85,B 0,C 180,E1 -21853.663,E2 -21853.663} C_VEL
LIN {X 0,Y 205.675,Z 450.072,A -85,B 0,C 180,E1 -21854.515,E2 -21854.515} C_VEL
LIN {X 0,Y 204.218,Z 462.15,A -85,B 0,C 180,E1 -21855.677,E2 -21855.677} C_VEL
LIN {X 0,Y 202.515,Z 473.859,A -85,B 0,C 180,E1 -21857.217,E2 -21857.217} C_VEL
LIN {X 0,Y 200.321,Z 485.635,A -85,B 0,C 180,E1 -21859.215,E2 -21859.215} C_VEL
LIN {X 0,Y 198.167,Z 495.434,A -85,B 0,C 180,E1 -21861.329,E2 -21861.329} C_VEL
LIN {X 0,Y 196.149,Z 504.607,A -85,B 0,C 180,E1 -21863.828,E2 -21863.828} C_VEL
LIN {X 0,Y 194.096,Z 513.553,A -85,B 0,C 180,E1 -21866.885,E2 -21866.885} C_VEL
LIN {X 0,Y 192.532,Z 520.737,A -85,B 0,C 180,E1 -21869.998,E2 -21869.998} C_VEL
LIN {X 0,Y 191.378,Z 526.46,A -85,B 0,C 180,E1 -21873.156,E2 -21873.156} C_VEL
LIN {X 0,Y 190.674,Z 530.965,A -85,B 0,C 180,E1 -21876.347,E2 -21876.347} C_VEL
LIN {X 0,Y 190.284,Z 533.357,A -85,B 0,C 180,E1 -21878.494,E2 -21878.494} C_VEL
LIN {X 0,Y 189.984,Z 535.32,A -85,B 0,C 180,E1 -21880.657,E2 -21880.657} C_VEL
LIN {X 0,Y 189.882,Z 536.822,A -85,B 0,C 180,E1 -21882.829,E2 -21882.829} C_VEL
LIN {X 0,Y 190.015,Z 538.229,A -85,B 0,C 180,E1 -21885.921,E2 -21885.921} C_VEL
LIN {X 0,Y 190.382,Z 538.802,A -85,B 0,C 180,E1 -21889.402,E2 -21889.402} C_VEL
LIN {X 0,Y 191.453,Z 538.125,A -85,B 0,C 180,E1 -21893.406,E2 -21893.406} C_VEL
LIN {X 0,Y 192.45,Z 536.956,A -85,B 0,C 180,E1 -21895.988,E2 -21895.988} C_VEL
LIN {X 0,Y 194.698,Z 533.851,A -85,B 0,C 180,E1 -21899.966,E2 -21899.966} C_VEL
LIN {X 0,Y 197.401,Z 529.64,A -85,B 0,C 180,E1 -21903.491,E2 -21903.491} C_VEL
LIN {X 0,Y 201.01,Z 523.603,A -85,B 0,C 180,E1 -21907.091,E2 -21907.091} C_VEL
LIN {X 0,Y 204.632,Z 516.831,A -85,B 0,C 180,E1 -21910.085,E2 -21910.085} C_VEL
LIN {X 0,Y 208.066,Z 509.883,A -85,B 0,C 180,E1 -21912.494,E2 -21912.494} C_VEL
LIN {X 0,Y 211.89,Z 501.439,A -85,B 0,C 180,E1 -21914.812,E2 -21914.812} C_VEL
LIN {X 0,Y 215.973,Z 491.23,A -85,B 0,C 180,E1 -21917.011,E2 -21917.011} C_VEL
LIN {X 0,Y 219.543,Z 480.586,A -85,B 0,C 180,E1 -21918.785,E2 -21918.785} C_VEL
LIN {X 0,Y 222.765,Z 469.101,A -85,B 0,C 180,E1 -21920.262,E2 -21920.262} C_VEL
LIN {X 0,Y 225.486,Z 456.907,A -85,B 0,C 180,E1 -21921.438,E2 -21921.438} C_VEL
LIN {X 0,Y 227.532,Z 443.422,A -85,B 0,C 180,E1 -21922.365,E2 -21922.365} C_VEL
LIN {X 0,Y 228.844,Z 430.701,A -85,B 0,C 180,E1 -21922.891,E2 -21922.891} C_VEL
LIN {X 0,Y 231.23,Z 391.614,A -85,B 0,C 180,E1 -21924.024,E2 -21924.024} C_VEL
LIN {X 0,Y 225.206,Z 378.936,A -85,B 0,C 180,E1 -21926.229,E2 -21926.229} C_VEL
LIN {X 0,Y 219.279,Z 368.001,A -85,B 0,C 180,E1 -21928.546,E2 -21928.546} C_VEL
LIN {X 0,Y 214.582,Z 360.434,A -85,B 0,C 180,E1 -21930.515,E2 -21930.515} C_VEL
LIN {X 0,Y 210.811,Z 355.338,A -85,B 0,C 180,E1 -21932.178,E2 -21932.178} C_VEL
LIN {X 0,Y 207.99,Z 351.488,A -85,B 0,C 180,E1 -21933.512,E2 -21933.512} C_VEL
LIN {X 0,Y 204.759,Z 347.209,A -85,B 0,C 180,E1 -21935.137,E2 -21935.137} C_VEL
LIN {X 0,Y 202.212,Z 344.168,A -85,B 0,C 180,E1 -21936.487,E2 -21936.487} C_VEL
LIN {X 0,Y 201.072,Z 342.403,A -85,B 0,C 180,E1 -21937.148,E2 -21937.148} C_VEL
LIN {X 0,Y 198.544,Z 339.941,A -85,B 0,C 180,E1 -21938.591,E2 -21938.591} C_VEL
LIN {X 0,Y 196.97,Z 337.192,A -85,B 0,C 180,E1 -21939.642,E2 -21939.642} C_VEL
LIN {X 0,Y 194.549,Z 335.47,A -85,B 0,C 180,E1 -21941.164,E2 -21941.164} C_VEL
LIN {X 0,Y 193.017,Z 332.925,A -85,B 0,C 180,E1 -21942.317,E2 -21942.317} C_VEL
LIN {X 0,Y 192.666,Z 331.472,A -85,B 0,C 180,E1 -21942.718,E2 -21942.718} C_VEL
LIN {X 0,Y 192.747,Z 331.459,A -85,B 0,C 180,E1 -21947.363,E2 -21947.363} C_VEL
LIN {X 0,Y 193.013,Z 331.422,A -85,B 0,C 180,E1 -21951.626,E2 -21951.626} C_VEL
LIN {X 0,Y 193.2,Z 331.403,A -85,B 0,C 180,E1 -21957.916,E2 -21957.916} C_VEL
LIN {X 0,Y 193.401,Z 331.392,A -85,B 0,C 180,E1 -21960,E2 -21960} C_VEL
LIN {X 0,Y 192.924,Z 331.445,A -85,B 0,C 180,E1 -21964.179,E2 -21964.179} C_VEL
LIN {X 0,Y 193.017,Z 331.42,A -85,B 0,C 180,E1 -21968.375,E2 -21968.375} C_VEL
LIN {X 0,Y 192.787,Z 331.448,A -85,B 0,C 180,E1 -21972.635,E2 -21972.635} C_VEL
LIN {X 0,Y 192.74,Z 331.46,A -85,B 0,C 180,E1 -21976.961,E2 -21976.961} C_VEL
LIN {X 0,Y 192.593,Z 331.486,A -85,B 0,C 180,E1 -21981.403,E2 -21981.403} C_VEL
LIN {X 0,Y 192.628,Z 331.477,A -85,B 0,C 180,E1 -21984.205,E2 -21984.205} C_VEL
LIN {X 0,Y 192.6,Z 331.564,A -85,B 0,C 180,E1 -21988.662,E2 -21988.662} C_VEL
LIN {X 0,Y 193.687,Z 334.495,A -85,B 0,C 180,E1 -21991.898,E2 -21991.898} C_VEL
LIN {X 0,Y 196.245,Z 338.439,A -85,B 0,C 180,E1 -21993.718,E2 -21993.718} C_VEL
LIN {X 0,Y 198.757,Z 341.422,A -85,B 0,C 180,E1 -21995.295,E2 -21995.295} C_VEL
LIN {X 0,Y 202.723,Z 346.855,A -85,B 0,C 180,E1 -21997.595,E2 -21997.595} C_VEL
LIN {X 0,Y 207.495,Z 354.127,A -85,B 0,C 180,E1 -22000.114,E2 -22000.114} C_VEL
LIN {X 0,Y 210.954,Z 359.51,A -85,B 0,C 180,E1 -22001.783,E2 -22001.783} C_VEL
LIN {X 0,Y 216.387,Z 368.546,A -85,B 0,C 180,E1 -22004.206,E2 -22004.206} C_VEL
LIN {X 0,Y 221.928,Z 378.893,A -85,B 0,C 180,E1 -22006.478,E2 -22006.478} C_VEL
LIN {X 0,Y 227.962,Z 391.973,A -85,B 0,C 180,E1 -22008.803,E2 -22008.803} C_VEL
LIN {X 0,Y 230.672,Z 398.807,A -85,B 0,C 180,E1 -22009.816,E2 -22009.816} C_VEL
LIN {X 0,Y 230.754,Z 402.391,A -85,B 0,C 180,E1 -22009.995,E2 -22009.995} C_VEL
LIN {X 0,Y 229.773,Z 417.816,A -85,B 0,C 180,E1 -22010.428,E2 -22010.428} C_VEL
LIN {X 0,Y 229.015,Z 423.666,A -85,B 0,C 180,E1 -22010.488,E2 -22010.488} C_VEL
LIN {X 0,Y 223.695,Z 442.703,A -85,B 0,C 180,E1 -22010.026,E2 -22010.026} C_VEL
LIN {X 0,Y 222.619,Z 448.507,A -85,B 0,C 180,E1 -22010.137,E2 -22010.137} C_VEL
LIN {X 0,Y 220.687,Z 461.365,A -85,B 0,C 180,E1 -22010.882,E2 -22010.882} C_VEL
LIN {X 0,Y 217.798,Z 473.897,A -85,B 0,C 180,E1 -22011.895,E2 -22011.895} C_VEL
LIN {X 0,Y 214.455,Z 485.884,A -85,B 0,C 180,E1 -22013.27,E2 -22013.27} C_VEL
LIN {X 0,Y 210.745,Z 496.625,A -85,B 0,C 180,E1 -22014.885,E2 -22014.885} C_VEL
LIN {X 0,Y 207.277,Z 505.419,A -85,B 0,C 180,E1 -22016.568,E2 -22016.568} C_VEL
LIN {X 0,Y 203.178,Z 514.483,A -85,B 0,C 180,E1 -22018.747,E2 -22018.747} C_VEL
LIN {X 0,Y 198.691,Z 523.34,A -85,B 0,C 180,E1 -22021.479,E2 -22021.479} C_VEL
LIN {X 0,Y 194.65,Z 530.82,A -85,B 0,C 180,E1 -22024.509,E2 -22024.509} C_VEL
